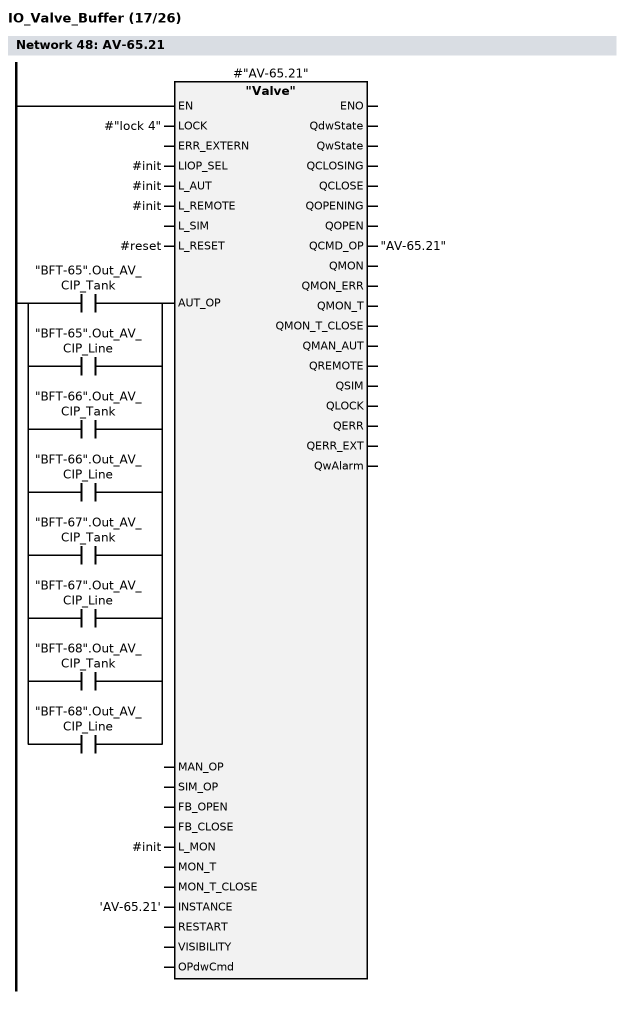
   RUNG wire#powerrail
      #"AV-65.21"(AUT_OP := wire#w1, LOCK := #"lock 4", ERR_EXTERN :=, LIOP_SEL := #init, L_AUT := #init, L_REMOTE := #init, L_SIM :=, L_RESET := #reset, MAN_OP :=, SIM_OP :=, FB_OPEN :=, FB_CLOSE :=, L_MON := #init, MON_T :=, MON_T_CLOSE :=, INSTANCE := 'AV-65.21', RESTART :=, VISIBILITY :=, OPdwCmd :=, QdwState =>, QwState =>, QCLOSING =>, QCLOSE =>, QOPENING =>, QOPEN =>, QCMD_OP => "AV-65.21", QMON =>, QMON_ERR =>, QMON_T =>, QMON_T_CLOSE =>, QMAN_AUT =>, QREMOTE =>, QSIM =>, QLOCK =>, QERR =>, QERR_EXT =>, QwAlarm =>)
   END_RUNG
   RUNG wire#powerrail
      Contact( "BFT-65".Out_AV_CIP_Tank )
   END_RUNG wire#w1
   RUNG wire#powerrail
      Contact( "BFT-65".Out_AV_CIP_Line )
   END_RUNG wire#w1
   RUNG wire#powerrail
      Contact( "BFT-66".Out_AV_CIP_Tank )
   END_RUNG wire#w1
   RUNG wire#powerrail
      Contact( "BFT-66".Out_AV_CIP_Line )
   END_RUNG wire#w1
   RUNG wire#powerrail
      Contact( "BFT-67".Out_AV_CIP_Tank )
   END_RUNG wire#w1
   RUNG wire#powerrail
      Contact( "BFT-67".Out_AV_CIP_Line )
   END_RUNG wire#w1
   RUNG wire#powerrail
      Contact( "BFT-68".Out_AV_CIP_Tank )
   END_RUNG wire#w1
   RUNG wire#powerrail
      Contact( "BFT-68".Out_AV_CIP_Line )
   END_RUNG wire#w1
   // the same network as SCL:
   #"AV-65.21"(LOCK := #"lock 4",   // "Valve"
               LIOP_SEL := #init,
               L_AUT := #init,
               L_REMOTE := #init,
               L_RESET := #reset,
               AUT_OP := "BFT-65".Out_AV_CIP_Tank OR "BFT-65".Out_AV_CIP_Line OR "BFT-66".Out_AV_CIP_Tank OR "BFT-66".Out_AV_CIP_Line OR "BFT-67".Out_AV_CIP_Tank OR "BFT-67".Out_AV_CIP_Line OR "BFT-68".Out_AV_CIP_Tank OR "BFT-68".Out_AV_CIP_Line,
               L_MON := #init,
               INSTANCE := 'AV-65.21',
               QCMD_OP => "AV-65.21");
END_REGION

REGION Network 50 (SCL): FB OPEN AND CLOSE VALVE T-66
   IF #testing THEN
       // Statement section IF
       #"AV-66.01".FB_OPEN := #"AV-66.01".QCMD_OP;
       #"AV-66.01".FB_CLOSE := NOT #"AV-66.01".QCMD_OP;
       #"AV-66.02".FB_OPEN := #"AV-66.02".QCMD_OP;
       #"AV-66.02".FB_CLOSE := NOT #"AV-66.02".QCMD_OP;
       #"AV-66.03".FB_OPEN := #"AV-66.03".QCMD_OP;
       #"AV-66.03".FB_CLOSE := NOT #"AV-66.03".QCMD_OP;
       #"AV-66.04".FB_OPEN := #"AV-66.04".QCMD_OP;
       #"AV-66.04".FB_CLOSE := NOT #"AV-66.04".QCMD_OP;
       #"AV-66.05".FB_OPEN := #"AV-66.05".QCMD_OP;
       #"AV-66.05".FB_CLOSE := NOT #"AV-66.05".QCMD_OP;
       #"AV-66.06".FB_OPEN := #"AV-66.06".QCMD_OP;
       #"AV-66.06".FB_CLOSE := NOT #"AV-66.06".QCMD_OP;
   ELSE
       // Statement section ELSE
       #"AV-66.01".FB_OPEN := NOT "ZSC-66.01";
       #"AV-66.01".FB_CLOSE := "ZSC-66.01";
       #"AV-66.02".FB_OPEN := #"AV-66.02".QCMD_OP;
       #"AV-66.02".FB_CLOSE := NOT #"AV-66.02".QCMD_OP;
       #"AV-66.03".FB_OPEN := NOT "ZSC-66.03";
       #"AV-66.03".FB_CLOSE := "ZSC-66.03";
       #"AV-66.04".FB_OPEN := #"AV-66.04".QCMD_OP;
       #"AV-66.04".FB_CLOSE := NOT #"AV-66.04".QCMD_OP;
       #"AV-66.05".FB_OPEN := #"AV-66.05".QCMD_OP;
       #"AV-66.05".FB_CLOSE := NOT #"AV-66.05".QCMD_OP;
       #"AV-66.06".FB_OPEN := NOT "ZSC-66.06";
       #"AV-66.06".FB_CLOSE := "ZSC-66.06";
   END_IF;
END_REGION

NETWORK
TITLE = FB MONITORING TIME VALVE T-66
// FB OPEN TIME
      L     T#20s;
      T     #"AV-66.01".MON_T;
      T     #"AV-66.02".MON_T;
      T     #"AV-66.03".MON_T;
      T     #"AV-66.04".MON_T;
      T     #"AV-66.05".MON_T;
      T     #"AV-66.06".MON_T;
// FB CLOSE TIME
      L     T#20s;
      T     #"AV-66.01".MON_T_CLOSE;
      T     #"AV-66.02".MON_T_CLOSE;
      T     #"AV-66.03".MON_T_CLOSE;
      T     #"AV-66.04".MON_T_CLOSE;
      T     #"AV-66.05".MON_T_CLOSE;
      T     #"AV-66.06".MON_T_CLOSE;

REGION Network 52: AV-66.01 w ZSC
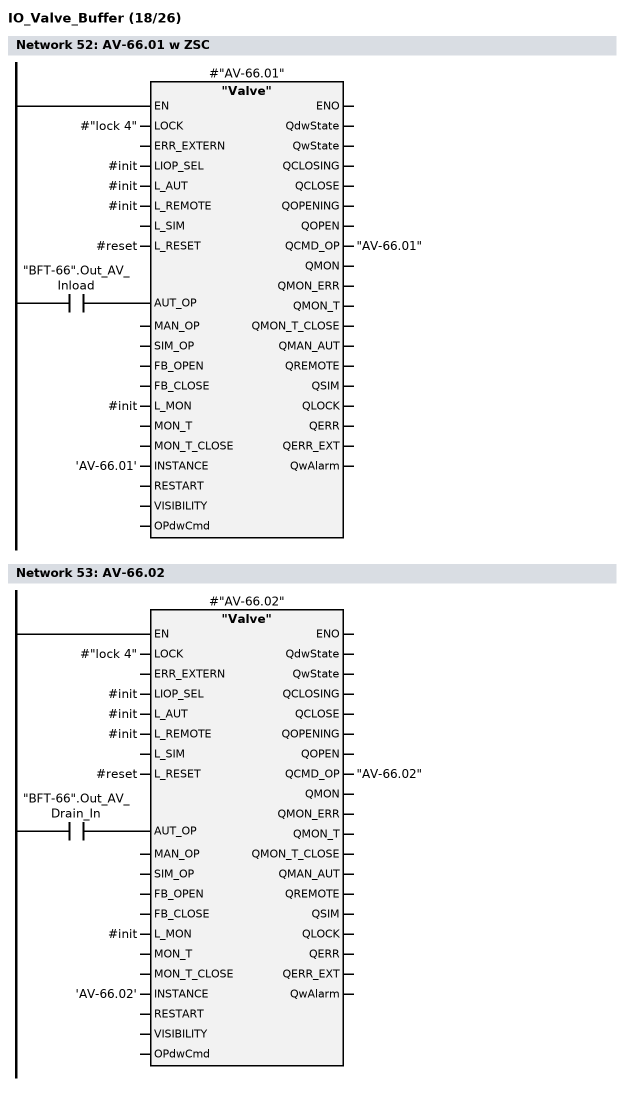
   RUNG wire#powerrail
      #"AV-66.01"(AUT_OP := wire#w1, LOCK := #"lock 4", ERR_EXTERN :=, LIOP_SEL := #init, L_AUT := #init, L_REMOTE := #init, L_SIM :=, L_RESET := #reset, MAN_OP :=, SIM_OP :=, FB_OPEN :=, FB_CLOSE :=, L_MON := #init, MON_T :=, MON_T_CLOSE :=, INSTANCE := 'AV-66.01', RESTART :=, VISIBILITY :=, OPdwCmd :=, QdwState =>, QwState =>, QCLOSING =>, QCLOSE =>, QOPENING =>, QOPEN =>, QCMD_OP => "AV-66.01", QMON =>, QMON_ERR =>, QMON_T =>, QMON_T_CLOSE =>, QMAN_AUT =>, QREMOTE =>, QSIM =>, QLOCK =>, QERR =>, QERR_EXT =>, QwAlarm =>)
   END_RUNG
   RUNG wire#powerrail
      Contact( "BFT-66".Out_AV_Inload )
   END_RUNG wire#w1
   // the same network as SCL:
   #"AV-66.01"(LOCK := #"lock 4",   // "Valve"
               LIOP_SEL := #init,
               L_AUT := #init,
               L_REMOTE := #init,
               L_RESET := #reset,
               AUT_OP := "BFT-66".Out_AV_Inload,
               L_MON := #init,
               INSTANCE := 'AV-66.01',
               QCMD_OP => "AV-66.01");
END_REGION

REGION Network 53: AV-66.02
   RUNG wire#powerrail
      #"AV-66.02"(AUT_OP := wire#w1, LOCK := #"lock 4", ERR_EXTERN :=, LIOP_SEL := #init, L_AUT := #init, L_REMOTE := #init, L_SIM :=, L_RESET := #reset, MAN_OP :=, SIM_OP :=, FB_OPEN :=, FB_CLOSE :=, L_MON := #init, MON_T :=, MON_T_CLOSE :=, INSTANCE := 'AV-66.02', RESTART :=, VISIBILITY :=, OPdwCmd :=, QdwState =>, QwState =>, QCLOSING =>, QCLOSE =>, QOPENING =>, QOPEN =>, QCMD_OP => "AV-66.02", QMON =>, QMON_ERR =>, QMON_T =>, QMON_T_CLOSE =>, QMAN_AUT =>, QREMOTE =>, QSIM =>, QLOCK =>, QERR =>, QERR_EXT =>, QwAlarm =>)
   END_RUNG
   RUNG wire#powerrail
      Contact( "BFT-66".Out_AV_Drain_In )
   END_RUNG wire#w1
   // the same network as SCL:
   #"AV-66.02"(LOCK := #"lock 4",   // "Valve"
               LIOP_SEL := #init,
               L_AUT := #init,
               L_REMOTE := #init,
               L_RESET := #reset,
               AUT_OP := "BFT-66".Out_AV_Drain_In,
               L_MON := #init,
               INSTANCE := 'AV-66.02',
               QCMD_OP => "AV-66.02");
END_REGION

REGION Network 54: AV-66.03 w ZSC
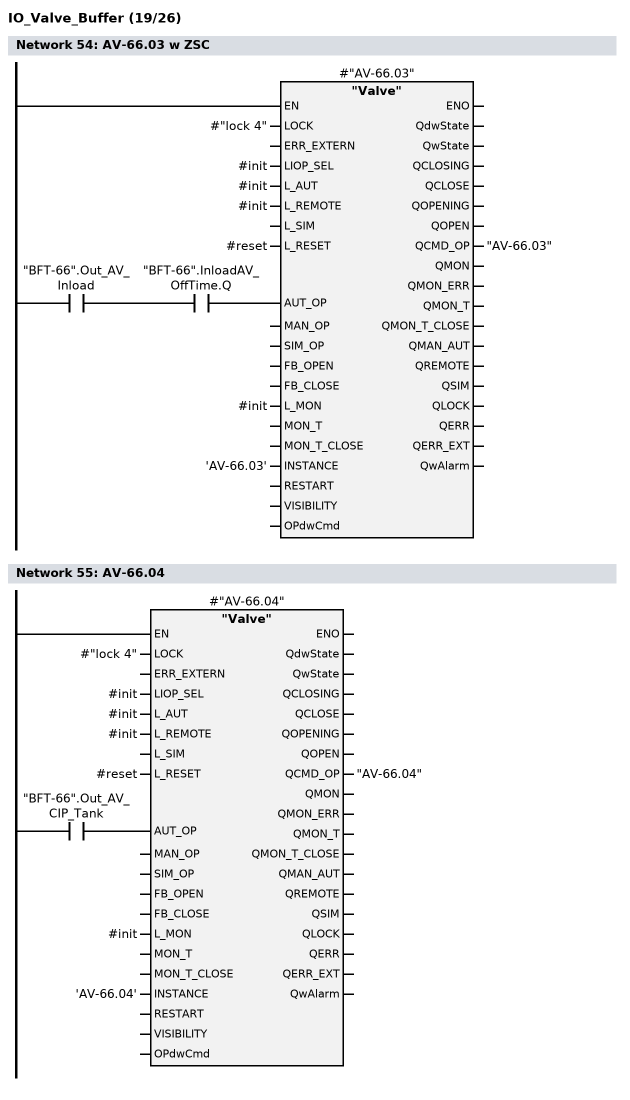
   RUNG wire#powerrail
      #"AV-66.03"(AUT_OP := wire#w1, LOCK := #"lock 4", ERR_EXTERN :=, LIOP_SEL := #init, L_AUT := #init, L_REMOTE := #init, L_SIM :=, L_RESET := #reset, MAN_OP :=, SIM_OP :=, FB_OPEN :=, FB_CLOSE :=, L_MON := #init, MON_T :=, MON_T_CLOSE :=, INSTANCE := 'AV-66.03', RESTART :=, VISIBILITY :=, OPdwCmd :=, QdwState =>, QwState =>, QCLOSING =>, QCLOSE =>, QOPENING =>, QOPEN =>, QCMD_OP => "AV-66.03", QMON =>, QMON_ERR =>, QMON_T =>, QMON_T_CLOSE =>, QMAN_AUT =>, QREMOTE =>, QSIM =>, QLOCK =>, QERR =>, QERR_EXT =>, QwAlarm =>)
   END_RUNG
   RUNG wire#powerrail
      Contact( "BFT-66".Out_AV_Inload )
      Contact( "BFT-66".InloadAV_OffTime.Q )
   END_RUNG wire#w1
   // the same network as SCL:
   #"AV-66.03"(LOCK := #"lock 4",   // "Valve"
               LIOP_SEL := #init,
               L_AUT := #init,
               L_REMOTE := #init,
               L_RESET := #reset,
               AUT_OP := "BFT-66".Out_AV_Inload AND "BFT-66".InloadAV_OffTime.Q,
               L_MON := #init,
               INSTANCE := 'AV-66.03',
               QCMD_OP => "AV-66.03");
END_REGION

REGION Network 55: AV-66.04
   RUNG wire#powerrail
      #"AV-66.04"(AUT_OP := wire#w1, LOCK := #"lock 4", ERR_EXTERN :=, LIOP_SEL := #init, L_AUT := #init, L_REMOTE := #init, L_SIM :=, L_RESET := #reset, MAN_OP :=, SIM_OP :=, FB_OPEN :=, FB_CLOSE :=, L_MON := #init, MON_T :=, MON_T_CLOSE :=, INSTANCE := 'AV-66.04', RESTART :=, VISIBILITY :=, OPdwCmd :=, QdwState =>, QwState =>, QCLOSING =>, QCLOSE =>, QOPENING =>, QOPEN =>, QCMD_OP => "AV-66.04", QMON =>, QMON_ERR =>, QMON_T =>, QMON_T_CLOSE =>, QMAN_AUT =>, QREMOTE =>, QSIM =>, QLOCK =>, QERR =>, QERR_EXT =>, QwAlarm =>)
   END_RUNG
   RUNG wire#powerrail
      Contact( "BFT-66".Out_AV_CIP_Tank )
   END_RUNG wire#w1
   // the same network as SCL:
   #"AV-66.04"(LOCK := #"lock 4",   // "Valve"
               LIOP_SEL := #init,
               L_AUT := #init,
               L_REMOTE := #init,
               L_RESET := #reset,
               AUT_OP := "BFT-66".Out_AV_CIP_Tank,
               L_MON := #init,
               INSTANCE := 'AV-66.04',
               QCMD_OP => "AV-66.04");
END_REGION

REGION Network 56: AV-66.05
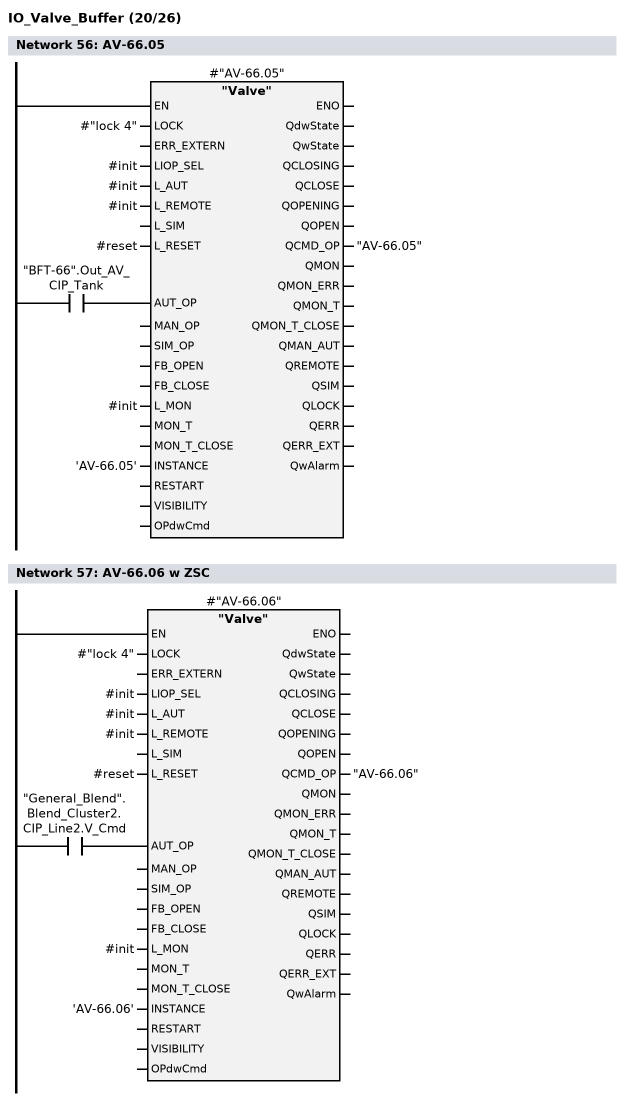
   RUNG wire#powerrail
      #"AV-66.05"(AUT_OP := wire#w1, LOCK := #"lock 4", ERR_EXTERN :=, LIOP_SEL := #init, L_AUT := #init, L_REMOTE := #init, L_SIM :=, L_RESET := #reset, MAN_OP :=, SIM_OP :=, FB_OPEN :=, FB_CLOSE :=, L_MON := #init, MON_T :=, MON_T_CLOSE :=, INSTANCE := 'AV-66.05', RESTART :=, VISIBILITY :=, OPdwCmd :=, QdwState =>, QwState =>, QCLOSING =>, QCLOSE =>, QOPENING =>, QOPEN =>, QCMD_OP => "AV-66.05", QMON =>, QMON_ERR =>, QMON_T =>, QMON_T_CLOSE =>, QMAN_AUT =>, QREMOTE =>, QSIM =>, QLOCK =>, QERR =>, QERR_EXT =>, QwAlarm =>)
   END_RUNG
   RUNG wire#powerrail
      Contact( "BFT-66".Out_AV_CIP_Tank )
   END_RUNG wire#w1
   // the same network as SCL:
   #"AV-66.05"(LOCK := #"lock 4",   // "Valve"
               LIOP_SEL := #init,
               L_AUT := #init,
               L_REMOTE := #init,
               L_RESET := #reset,
               AUT_OP := "BFT-66".Out_AV_CIP_Tank,
               L_MON := #init,
               INSTANCE := 'AV-66.05',
               QCMD_OP => "AV-66.05");
END_REGION

REGION Network 57: AV-66.06 w ZSC
   RUNG wire#powerrail
      #"AV-66.06"(AUT_OP := wire#w1, LOCK := #"lock 4", ERR_EXTERN :=, LIOP_SEL := #init, L_AUT := #init, L_REMOTE := #init, L_SIM :=, L_RESET := #reset, MAN_OP :=, SIM_OP :=, FB_OPEN :=, FB_CLOSE :=, L_MON := #init, MON_T :=, MON_T_CLOSE :=, INSTANCE := 'AV-66.06', RESTART :=, VISIBILITY :=, OPdwCmd :=, QdwState =>, QwState =>, QCLOSING =>, QCLOSE =>, QOPENING =>, QOPEN =>, QCMD_OP => "AV-66.06", QMON =>, QMON_ERR =>, QMON_T =>, QMON_T_CLOSE =>, QMAN_AUT =>, QREMOTE =>, QSIM =>, QLOCK =>, QERR =>, QERR_EXT =>, QwAlarm =>)
   END_RUNG
   RUNG wire#powerrail
      Contact( "General_Blend".Blend_Cluster2.CIP_Line2.V_Cmd )
   END_RUNG wire#w1
   // the same network as SCL:
   #"AV-66.06"(LOCK := #"lock 4",   // "Valve"
               LIOP_SEL := #init,
               L_AUT := #init,
               L_REMOTE := #init,
               L_RESET := #reset,
               AUT_OP := "General_Blend".Blend_Cluster2.CIP_Line2.V_Cmd,
               L_MON := #init,
               INSTANCE := 'AV-66.06',
               QCMD_OP => "AV-66.06");
END_REGION

REGION Network 59 (SCL): FB OPEN AND CLOSE VALVE T-67
   IF #testing THEN
       // Statement section IF
       #"AV-67.01".FB_OPEN := #"AV-67.01".QCMD_OP;
       #"AV-67.01".FB_CLOSE := NOT #"AV-67.01".QCMD_OP;
       #"AV-67.02".FB_OPEN := #"AV-67.02".QCMD_OP;
       #"AV-67.02".FB_CLOSE := NOT #"AV-67.02".QCMD_OP;
       #"AV-67.03".FB_OPEN := #"AV-67.03".QCMD_OP;
       #"AV-67.03".FB_CLOSE := NOT #"AV-67.03".QCMD_OP;
       #"AV-67.04".FB_OPEN := #"AV-67.04".QCMD_OP;
       #"AV-67.04".FB_CLOSE := NOT #"AV-67.04".QCMD_OP;
       #"AV-67.05".FB_OPEN := #"AV-67.05".QCMD_OP;
       #"AV-67.05".FB_CLOSE := NOT #"AV-67.05".QCMD_OP;
   ELSE
       // Statement section ELSE
       #"AV-67.01".FB_OPEN := NOT "ZSC-67.01";
       #"AV-67.01".FB_CLOSE := "ZSC-67.01";
       #"AV-67.02".FB_OPEN := #"AV-67.02".QCMD_OP;
       #"AV-67.02".FB_CLOSE := NOT #"AV-67.02".QCMD_OP;
       #"AV-67.03".FB_OPEN := NOT "ZSC-67.03";
       #"AV-67.03".FB_CLOSE := "ZSC-67.03";
       #"AV-67.04".FB_OPEN := #"AV-67.04".QCMD_OP;
       #"AV-67.04".FB_CLOSE := NOT #"AV-67.04".QCMD_OP;
       #"AV-67.05".FB_OPEN := #"AV-67.05".QCMD_OP;
       #"AV-67.05".FB_CLOSE := NOT #"AV-67.05".QCMD_OP;
   END_IF;
END_REGION

NETWORK
TITLE = FB MONITORING TIME VALVE T-67
// FB OPEN TIME
      L     T#20s;
      T     #"AV-67.01".MON_T;
      T     #"AV-67.02".MON_T;
      T     #"AV-67.03".MON_T;
      T     #"AV-67.04".MON_T;
      T     #"AV-67.05".MON_T;
// FB CLOSE TIME
      L     T#20s;
      T     #"AV-67.01".MON_T_CLOSE;
      T     #"AV-67.02".MON_T_CLOSE;
      T     #"AV-67.03".MON_T_CLOSE;
      T     #"AV-67.04".MON_T_CLOSE;
      T     #"AV-67.05".MON_T_CLOSE;


REGION Network 61: AV-67.01 w ZSC
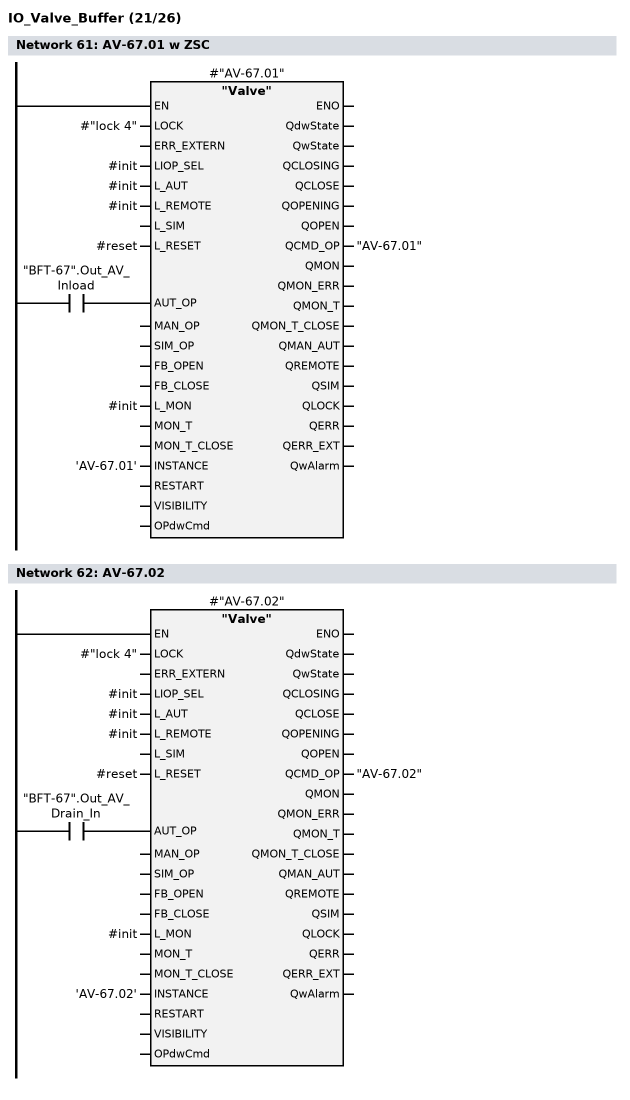
   RUNG wire#powerrail
      #"AV-67.01"(AUT_OP := wire#w1, LOCK := #"lock 4", ERR_EXTERN :=, LIOP_SEL := #init, L_AUT := #init, L_REMOTE := #init, L_SIM :=, L_RESET := #reset, MAN_OP :=, SIM_OP :=, FB_OPEN :=, FB_CLOSE :=, L_MON := #init, MON_T :=, MON_T_CLOSE :=, INSTANCE := 'AV-67.01', RESTART :=, VISIBILITY :=, OPdwCmd :=, QdwState =>, QwState =>, QCLOSING =>, QCLOSE =>, QOPENING =>, QOPEN =>, QCMD_OP => "AV-67.01", QMON =>, QMON_ERR =>, QMON_T =>, QMON_T_CLOSE =>, QMAN_AUT =>, QREMOTE =>, QSIM =>, QLOCK =>, QERR =>, QERR_EXT =>, QwAlarm =>)
   END_RUNG
   RUNG wire#powerrail
      Contact( "BFT-67".Out_AV_Inload )
   END_RUNG wire#w1
   // the same network as SCL:
   #"AV-67.01"(LOCK := #"lock 4",   // "Valve"
               LIOP_SEL := #init,
               L_AUT := #init,
               L_REMOTE := #init,
               L_RESET := #reset,
               AUT_OP := "BFT-67".Out_AV_Inload,
               L_MON := #init,
               INSTANCE := 'AV-67.01',
               QCMD_OP => "AV-67.01");
END_REGION

REGION Network 62: AV-67.02
   RUNG wire#powerrail
      #"AV-67.02"(AUT_OP := wire#w1, LOCK := #"lock 4", ERR_EXTERN :=, LIOP_SEL := #init, L_AUT := #init, L_REMOTE := #init, L_SIM :=, L_RESET := #reset, MAN_OP :=, SIM_OP :=, FB_OPEN :=, FB_CLOSE :=, L_MON := #init, MON_T :=, MON_T_CLOSE :=, INSTANCE := 'AV-67.02', RESTART :=, VISIBILITY :=, OPdwCmd :=, QdwState =>, QwState =>, QCLOSING =>, QCLOSE =>, QOPENING =>, QOPEN =>, QCMD_OP => "AV-67.02", QMON =>, QMON_ERR =>, QMON_T =>, QMON_T_CLOSE =>, QMAN_AUT =>, QREMOTE =>, QSIM =>, QLOCK =>, QERR =>, QERR_EXT =>, QwAlarm =>)
   END_RUNG
   RUNG wire#powerrail
      Contact( "BFT-67".Out_AV_Drain_In )
   END_RUNG wire#w1
   // the same network as SCL:
   #"AV-67.02"(LOCK := #"lock 4",   // "Valve"
               LIOP_SEL := #init,
               L_AUT := #init,
               L_REMOTE := #init,
               L_RESET := #reset,
               AUT_OP := "BFT-67".Out_AV_Drain_In,
               L_MON := #init,
               INSTANCE := 'AV-67.02',
               QCMD_OP => "AV-67.02");
END_REGION

REGION Network 63: AV-67.03 w ZSC
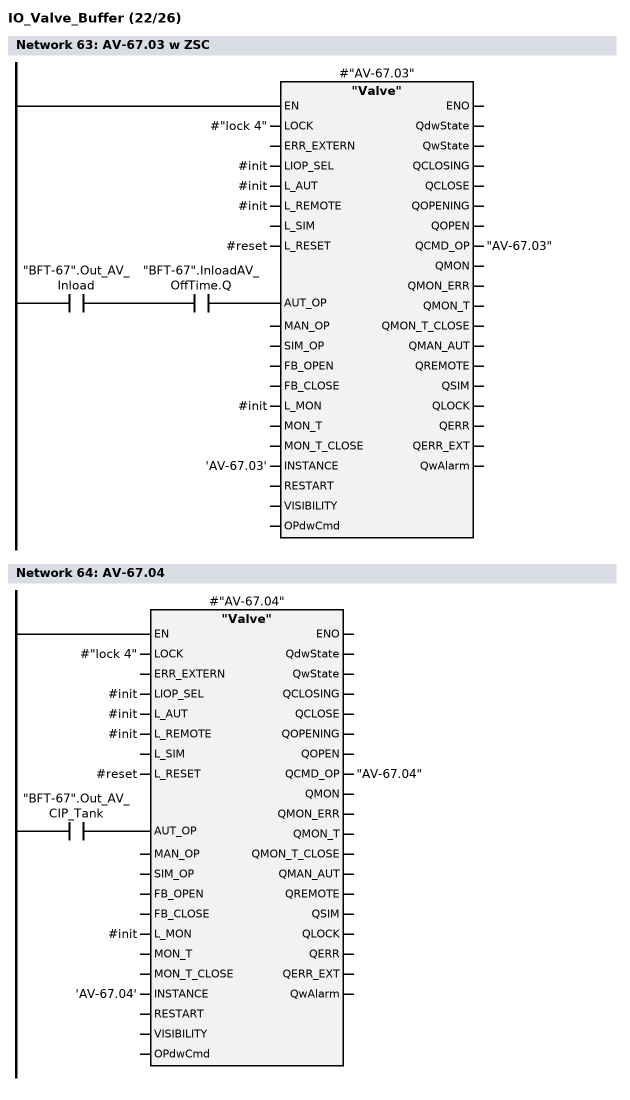
   RUNG wire#powerrail
      #"AV-67.03"(AUT_OP := wire#w1, LOCK := #"lock 4", ERR_EXTERN :=, LIOP_SEL := #init, L_AUT := #init, L_REMOTE := #init, L_SIM :=, L_RESET := #reset, MAN_OP :=, SIM_OP :=, FB_OPEN :=, FB_CLOSE :=, L_MON := #init, MON_T :=, MON_T_CLOSE :=, INSTANCE := 'AV-67.03', RESTART :=, VISIBILITY :=, OPdwCmd :=, QdwState =>, QwState =>, QCLOSING =>, QCLOSE =>, QOPENING =>, QOPEN =>, QCMD_OP => "AV-67.03", QMON =>, QMON_ERR =>, QMON_T =>, QMON_T_CLOSE =>, QMAN_AUT =>, QREMOTE =>, QSIM =>, QLOCK =>, QERR =>, QERR_EXT =>, QwAlarm =>)
   END_RUNG
   RUNG wire#powerrail
      Contact( "BFT-67".Out_AV_Inload )
      Contact( "BFT-67".InloadAV_OffTime.Q )
   END_RUNG wire#w1
   // the same network as SCL:
   #"AV-67.03"(LOCK := #"lock 4",   // "Valve"
               LIOP_SEL := #init,
               L_AUT := #init,
               L_REMOTE := #init,
               L_RESET := #reset,
               AUT_OP := "BFT-67".Out_AV_Inload AND "BFT-67".InloadAV_OffTime.Q,
               L_MON := #init,
               INSTANCE := 'AV-67.03',
               QCMD_OP => "AV-67.03");
END_REGION

REGION Network 64: AV-67.04
   RUNG wire#powerrail
      #"AV-67.04"(AUT_OP := wire#w1, LOCK := #"lock 4", ERR_EXTERN :=, LIOP_SEL := #init, L_AUT := #init, L_REMOTE := #init, L_SIM :=, L_RESET := #reset, MAN_OP :=, SIM_OP :=, FB_OPEN :=, FB_CLOSE :=, L_MON := #init, MON_T :=, MON_T_CLOSE :=, INSTANCE := 'AV-67.04', RESTART :=, VISIBILITY :=, OPdwCmd :=, QdwState =>, QwState =>, QCLOSING =>, QCLOSE =>, QOPENING =>, QOPEN =>, QCMD_OP => "AV-67.04", QMON =>, QMON_ERR =>, QMON_T =>, QMON_T_CLOSE =>, QMAN_AUT =>, QREMOTE =>, QSIM =>, QLOCK =>, QERR =>, QERR_EXT =>, QwAlarm =>)
   END_RUNG
   RUNG wire#powerrail
      Contact( "BFT-67".Out_AV_CIP_Tank )
   END_RUNG wire#w1
   // the same network as SCL:
   #"AV-67.04"(LOCK := #"lock 4",   // "Valve"
               LIOP_SEL := #init,
               L_AUT := #init,
               L_REMOTE := #init,
               L_RESET := #reset,
               AUT_OP := "BFT-67".Out_AV_CIP_Tank,
               L_MON := #init,
               INSTANCE := 'AV-67.04',
               QCMD_OP => "AV-67.04");
END_REGION

REGION Network 65: AV-67.05
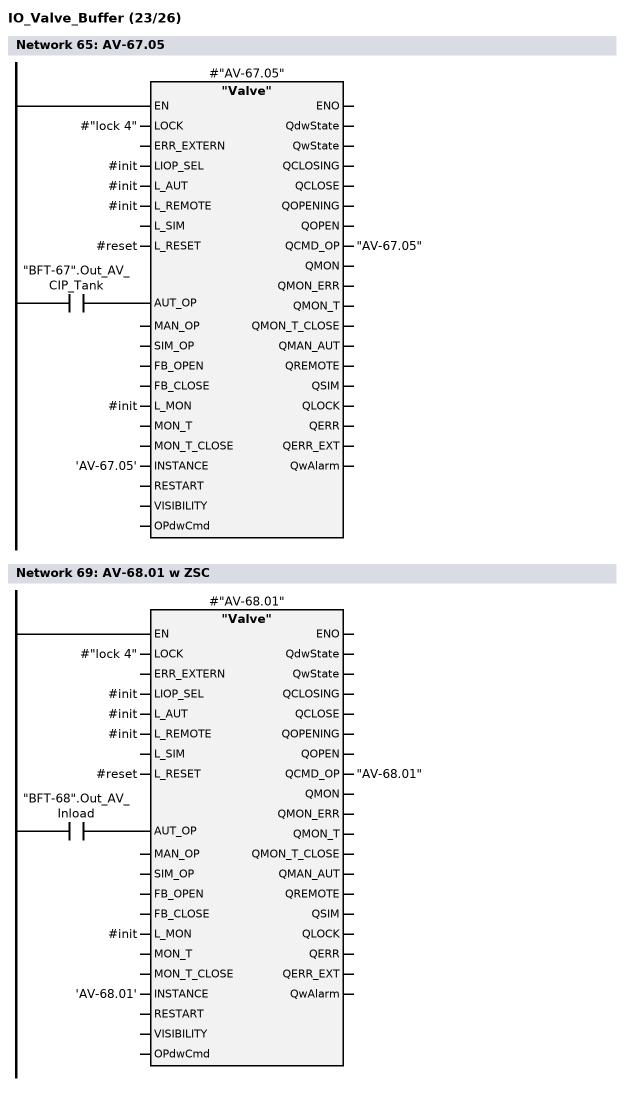
   RUNG wire#powerrail
      #"AV-67.05"(AUT_OP := wire#w1, LOCK := #"lock 4", ERR_EXTERN :=, LIOP_SEL := #init, L_AUT := #init, L_REMOTE := #init, L_SIM :=, L_RESET := #reset, MAN_OP :=, SIM_OP :=, FB_OPEN :=, FB_CLOSE :=, L_MON := #init, MON_T :=, MON_T_CLOSE :=, INSTANCE := 'AV-67.05', RESTART :=, VISIBILITY :=, OPdwCmd :=, QdwState =>, QwState =>, QCLOSING =>, QCLOSE =>, QOPENING =>, QOPEN =>, QCMD_OP => "AV-67.05", QMON =>, QMON_ERR =>, QMON_T =>, QMON_T_CLOSE =>, QMAN_AUT =>, QREMOTE =>, QSIM =>, QLOCK =>, QERR =>, QERR_EXT =>, QwAlarm =>)
   END_RUNG
   RUNG wire#powerrail
      Contact( "BFT-67".Out_AV_CIP_Tank )
   END_RUNG wire#w1
   // the same network as SCL:
   #"AV-67.05"(LOCK := #"lock 4",   // "Valve"
               LIOP_SEL := #init,
               L_AUT := #init,
               L_REMOTE := #init,
               L_RESET := #reset,
               AUT_OP := "BFT-67".Out_AV_CIP_Tank,
               L_MON := #init,
               INSTANCE := 'AV-67.05',
               QCMD_OP => "AV-67.05");
END_REGION

REGION Network 67 (SCL): FB OPEN AND CLOSE VALVE T-68
   IF #testing THEN
       // Statement section IF
       #"AV-68.01".FB_OPEN := #"AV-68.01".QCMD_OP;
       #"AV-68.01".FB_CLOSE := NOT #"AV-68.01".QCMD_OP;
       #"AV-68.02".FB_OPEN := #"AV-68.02".QCMD_OP;
       #"AV-68.02".FB_CLOSE := NOT #"AV-68.02".QCMD_OP;
       #"AV-68.03".FB_OPEN := #"AV-68.03".QCMD_OP;
       #"AV-68.03".FB_CLOSE := NOT #"AV-68.03".QCMD_OP;
       #"AV-68.04".FB_OPEN := #"AV-68.04".QCMD_OP;
       #"AV-68.04".FB_CLOSE := NOT #"AV-68.04".QCMD_OP;
       #"AV-68.05".FB_OPEN := #"AV-68.05".QCMD_OP;
       #"AV-68.05".FB_CLOSE := NOT #"AV-68.05".QCMD_OP;
       #"AV-68.06".FB_OPEN := #"AV-68.06".QCMD_OP;
       #"AV-68.06".FB_CLOSE := NOT #"AV-68.06".QCMD_OP;
   ELSE
       // Statement section ELSE
       #"AV-68.01".FB_OPEN := NOT "ZSC-68.01";
       #"AV-68.01".FB_CLOSE := "ZSC-68.01";
       #"AV-68.02".FB_OPEN := #"AV-68.02".QCMD_OP;
       #"AV-68.02".FB_CLOSE := NOT #"AV-68.02".QCMD_OP;
       #"AV-68.03".FB_OPEN := NOT "ZSC-68.03";
       #"AV-68.03".FB_CLOSE := "ZSC-68.03";
       #"AV-68.04".FB_OPEN := #"AV-68.04".QCMD_OP;
       #"AV-68.04".FB_CLOSE := NOT #"AV-68.04".QCMD_OP;
       #"AV-68.05".FB_OPEN := #"AV-68.05".QCMD_OP;
       #"AV-68.05".FB_CLOSE := NOT #"AV-68.05".QCMD_OP;
       #"AV-68.06".FB_OPEN := NOT "ZSC-68.06";
       #"AV-68.06".FB_CLOSE := "ZSC-68.06";
   END_IF;
END_REGION

NETWORK
TITLE = FB MONITORING TIME VALVE T-68
// FB OPEN TIME
      L     T#20s;
      T     #"AV-68.01".MON_T;
      T     #"AV-68.02".MON_T;
      T     #"AV-68.03".MON_T;
      T     #"AV-68.04".MON_T;
      T     #"AV-68.05".MON_T;
      T     #"AV-68.06".MON_T;
// FB CLOSE TIME
      L     T#20s;
      T     #"AV-68.01".MON_T_CLOSE;
      T     #"AV-68.02".MON_T_CLOSE;
      T     #"AV-68.03".MON_T_CLOSE;
      T     #"AV-68.04".MON_T_CLOSE;
      T     #"AV-68.05".MON_T_CLOSE;
      T     #"AV-68.06".MON_T_CLOSE;

REGION Network 69: AV-68.01 w ZSC
   RUNG wire#powerrail
      #"AV-68.01"(AUT_OP := wire#w1, LOCK := #"lock 4", ERR_EXTERN :=, LIOP_SEL := #init, L_AUT := #init, L_REMOTE := #init, L_SIM :=, L_RESET := #reset, MAN_OP :=, SIM_OP :=, FB_OPEN :=, FB_CLOSE :=, L_MON := #init, MON_T :=, MON_T_CLOSE :=, INSTANCE := 'AV-68.01', RESTART :=, VISIBILITY :=, OPdwCmd :=, QdwState =>, QwState =>, QCLOSING =>, QCLOSE =>, QOPENING =>, QOPEN =>, QCMD_OP => "AV-68.01", QMON =>, QMON_ERR =>, QMON_T =>, QMON_T_CLOSE =>, QMAN_AUT =>, QREMOTE =>, QSIM =>, QLOCK =>, QERR =>, QERR_EXT =>, QwAlarm =>)
   END_RUNG
   RUNG wire#powerrail
      Contact( "BFT-68".Out_AV_Inload )
   END_RUNG wire#w1
   // the same network as SCL:
   #"AV-68.01"(LOCK := #"lock 4",   // "Valve"
               LIOP_SEL := #init,
               L_AUT := #init,
               L_REMOTE := #init,
               L_RESET := #reset,
               AUT_OP := "BFT-68".Out_AV_Inload,
               L_MON := #init,
               INSTANCE := 'AV-68.01',
               QCMD_OP => "AV-68.01");
END_REGION

REGION Network 70: AV-68.02
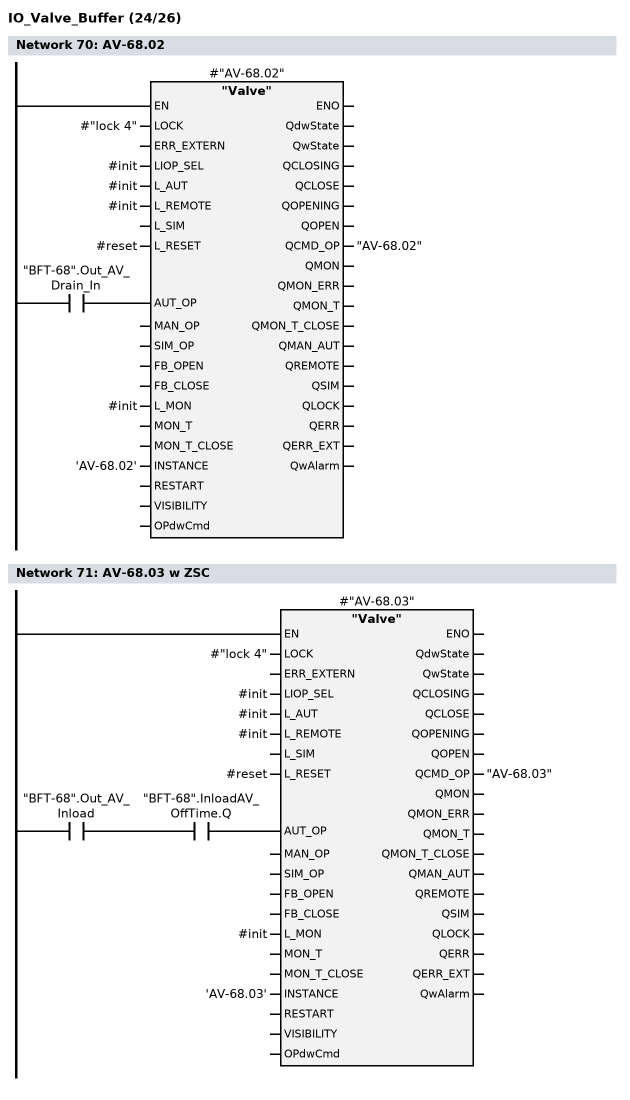
   RUNG wire#powerrail
      #"AV-68.02"(AUT_OP := wire#w1, LOCK := #"lock 4", ERR_EXTERN :=, LIOP_SEL := #init, L_AUT := #init, L_REMOTE := #init, L_SIM :=, L_RESET := #reset, MAN_OP :=, SIM_OP :=, FB_OPEN :=, FB_CLOSE :=, L_MON := #init, MON_T :=, MON_T_CLOSE :=, INSTANCE := 'AV-68.02', RESTART :=, VISIBILITY :=, OPdwCmd :=, QdwState =>, QwState =>, QCLOSING =>, QCLOSE =>, QOPENING =>, QOPEN =>, QCMD_OP => "AV-68.02", QMON =>, QMON_ERR =>, QMON_T =>, QMON_T_CLOSE =>, QMAN_AUT =>, QREMOTE =>, QSIM =>, QLOCK =>, QERR =>, QERR_EXT =>, QwAlarm =>)
   END_RUNG
   RUNG wire#powerrail
      Contact( "BFT-68".Out_AV_Drain_In )
   END_RUNG wire#w1
   // the same network as SCL:
   #"AV-68.02"(LOCK := #"lock 4",   // "Valve"
               LIOP_SEL := #init,
               L_AUT := #init,
               L_REMOTE := #init,
               L_RESET := #reset,
               AUT_OP := "BFT-68".Out_AV_Drain_In,
               L_MON := #init,
               INSTANCE := 'AV-68.02',
               QCMD_OP => "AV-68.02");
END_REGION

REGION Network 71: AV-68.03 w ZSC
   RUNG wire#powerrail
      #"AV-68.03"(AUT_OP := wire#w1, LOCK := #"lock 4", ERR_EXTERN :=, LIOP_SEL := #init, L_AUT := #init, L_REMOTE := #init, L_SIM :=, L_RESET := #reset, MAN_OP :=, SIM_OP :=, FB_OPEN :=, FB_CLOSE :=, L_MON := #init, MON_T :=, MON_T_CLOSE :=, INSTANCE := 'AV-68.03', RESTART :=, VISIBILITY :=, OPdwCmd :=, QdwState =>, QwState =>, QCLOSING =>, QCLOSE =>, QOPENING =>, QOPEN =>, QCMD_OP => "AV-68.03", QMON =>, QMON_ERR =>, QMON_T =>, QMON_T_CLOSE =>, QMAN_AUT =>, QREMOTE =>, QSIM =>, QLOCK =>, QERR =>, QERR_EXT =>, QwAlarm =>)
   END_RUNG
   RUNG wire#powerrail
      Contact( "BFT-68".Out_AV_Inload )
      Contact( "BFT-68".InloadAV_OffTime.Q )
   END_RUNG wire#w1
   // the same network as SCL:
   #"AV-68.03"(LOCK := #"lock 4",   // "Valve"
               LIOP_SEL := #init,
               L_AUT := #init,
               L_REMOTE := #init,
               L_RESET := #reset,
               AUT_OP := "BFT-68".Out_AV_Inload AND "BFT-68".InloadAV_OffTime.Q,
               L_MON := #init,
               INSTANCE := 'AV-68.03',
               QCMD_OP => "AV-68.03");
END_REGION

REGION Network 72: AV-68.04
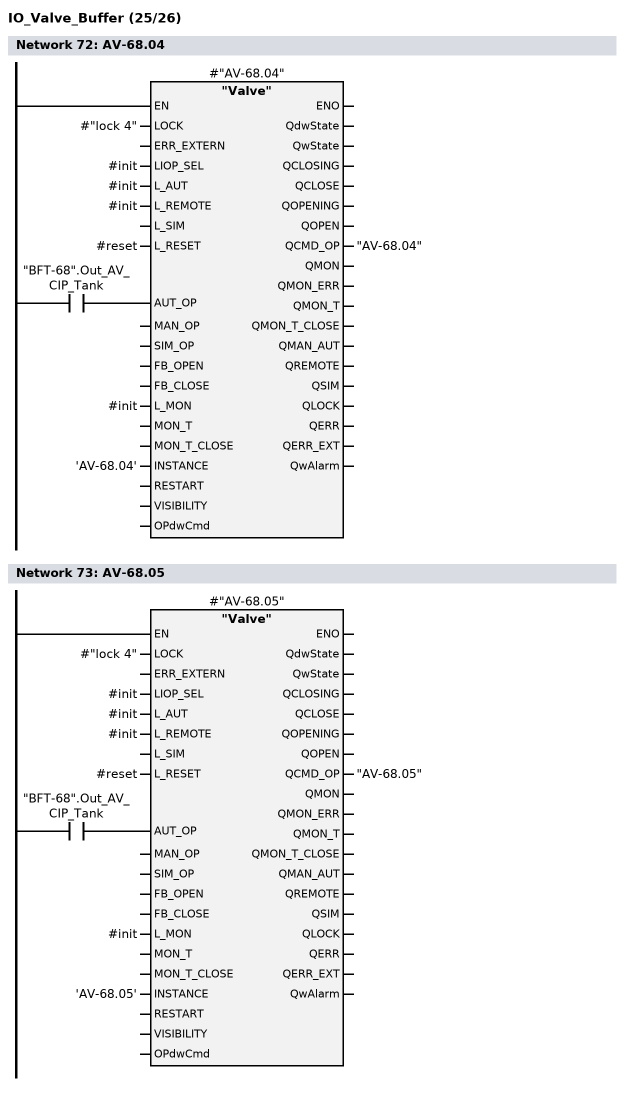
   RUNG wire#powerrail
      #"AV-68.04"(AUT_OP := wire#w1, LOCK := #"lock 4", ERR_EXTERN :=, LIOP_SEL := #init, L_AUT := #init, L_REMOTE := #init, L_SIM :=, L_RESET := #reset, MAN_OP :=, SIM_OP :=, FB_OPEN :=, FB_CLOSE :=, L_MON := #init, MON_T :=, MON_T_CLOSE :=, INSTANCE := 'AV-68.04', RESTART :=, VISIBILITY :=, OPdwCmd :=, QdwState =>, QwState =>, QCLOSING =>, QCLOSE =>, QOPENING =>, QOPEN =>, QCMD_OP => "AV-68.04", QMON =>, QMON_ERR =>, QMON_T =>, QMON_T_CLOSE =>, QMAN_AUT =>, QREMOTE =>, QSIM =>, QLOCK =>, QERR =>, QERR_EXT =>, QwAlarm =>)
   END_RUNG
   RUNG wire#powerrail
      Contact( "BFT-68".Out_AV_CIP_Tank )
   END_RUNG wire#w1
   // the same network as SCL:
   #"AV-68.04"(LOCK := #"lock 4",   // "Valve"
               LIOP_SEL := #init,
               L_AUT := #init,
               L_REMOTE := #init,
               L_RESET := #reset,
               AUT_OP := "BFT-68".Out_AV_CIP_Tank,
               L_MON := #init,
               INSTANCE := 'AV-68.04',
               QCMD_OP => "AV-68.04");
END_REGION

REGION Network 73: AV-68.05
   RUNG wire#powerrail
      #"AV-68.05"(AUT_OP := wire#w1, LOCK := #"lock 4", ERR_EXTERN :=, LIOP_SEL := #init, L_AUT := #init, L_REMOTE := #init, L_SIM :=, L_RESET := #reset, MAN_OP :=, SIM_OP :=, FB_OPEN :=, FB_CLOSE :=, L_MON := #init, MON_T :=, MON_T_CLOSE :=, INSTANCE := 'AV-68.05', RESTART :=, VISIBILITY :=, OPdwCmd :=, QdwState =>, QwState =>, QCLOSING =>, QCLOSE =>, QOPENING =>, QOPEN =>, QCMD_OP => "AV-68.05", QMON =>, QMON_ERR =>, QMON_T =>, QMON_T_CLOSE =>, QMAN_AUT =>, QREMOTE =>, QSIM =>, QLOCK =>, QERR =>, QERR_EXT =>, QwAlarm =>)
   END_RUNG
   RUNG wire#powerrail
      Contact( "BFT-68".Out_AV_CIP_Tank )
   END_RUNG wire#w1
   // the same network as SCL:
   #"AV-68.05"(LOCK := #"lock 4",   // "Valve"
               LIOP_SEL := #init,
               L_AUT := #init,
               L_REMOTE := #init,
               L_RESET := #reset,
               AUT_OP := "BFT-68".Out_AV_CIP_Tank,
               L_MON := #init,
               INSTANCE := 'AV-68.05',
               QCMD_OP => "AV-68.05");
END_REGION

REGION Network 74: AV-68.06 w ZSC
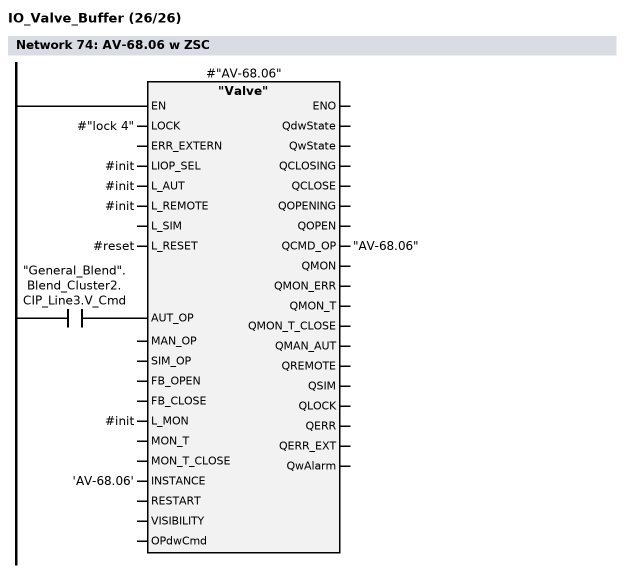
   RUNG wire#powerrail
      #"AV-68.06"(AUT_OP := wire#w1, LOCK := #"lock 4", ERR_EXTERN :=, LIOP_SEL := #init, L_AUT := #init, L_REMOTE := #init, L_SIM :=, L_RESET := #reset, MAN_OP :=, SIM_OP :=, FB_OPEN :=, FB_CLOSE :=, L_MON := #init, MON_T :=, MON_T_CLOSE :=, INSTANCE := 'AV-68.06', RESTART :=, VISIBILITY :=, OPdwCmd :=, QdwState =>, QwState =>, QCLOSING =>, QCLOSE =>, QOPENING =>, QOPEN =>, QCMD_OP => "AV-68.06", QMON =>, QMON_ERR =>, QMON_T =>, QMON_T_CLOSE =>, QMAN_AUT =>, QREMOTE =>, QSIM =>, QLOCK =>, QERR =>, QERR_EXT =>, QwAlarm =>)
   END_RUNG
   RUNG wire#powerrail
      Contact( "General_Blend".Blend_Cluster2.CIP_Line3.V_Cmd )
   END_RUNG wire#w1
   // the same network as SCL:
   #"AV-68.06"(LOCK := #"lock 4",   // "Valve"
               LIOP_SEL := #init,
               L_AUT := #init,
               L_REMOTE := #init,
               L_RESET := #reset,
               AUT_OP := "General_Blend".Blend_Cluster2.CIP_Line3.V_Cmd,
               L_MON := #init,
               INSTANCE := 'AV-68.06',
               QCMD_OP => "AV-68.06");
END_REGION
END_FUNCTION_BLOCK

FUNCTION_BLOCK "Alarm_Collector_Gen"   // FB33, LAD
{ S7_Optimized_Access := 'TRUE' }
VERSION : 0.1
// stored: AutoNumber true, IsIECCheckEnabled false, IsRetainMemResEnabled false, MemoryReserve 100, SetENOAutomatically false, UDAEnableTagReadback false
   VAR
      Alarm_DRP : DWord;   // Dry Run Protection Alarm
      Alarm_PS : DWord;   // Pressure Switch Alarm
   END_VAR
BEGIN

REGION Network 1: Alarm DRP
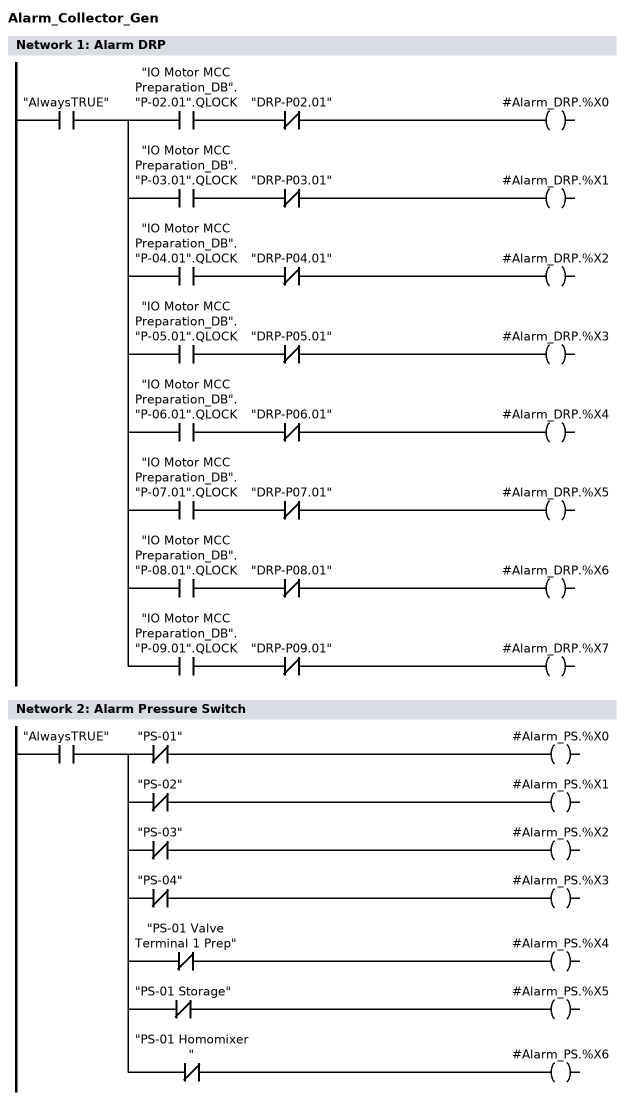
   RUNG wire#powerrail
      Contact( "AlwaysTRUE" )
      wire#w1
      Contact( "IO Motor MCC Preparation_DB"."P-02.01".QLOCK )
      I_Contact( "DRP-P02.01" )
      Coil( #Alarm_DRP.%X0 )
   END_RUNG
   RUNG wire#w1
      Contact( "IO Motor MCC Preparation_DB"."P-03.01".QLOCK )
      I_Contact( "DRP-P03.01" )
      Coil( #Alarm_DRP.%X1 )
   END_RUNG
   RUNG wire#w1
      Contact( "IO Motor MCC Preparation_DB"."P-04.01".QLOCK )
      I_Contact( "DRP-P04.01" )
      Coil( #Alarm_DRP.%X2 )
   END_RUNG
   RUNG wire#w1
      Contact( "IO Motor MCC Preparation_DB"."P-05.01".QLOCK )
      I_Contact( "DRP-P05.01" )
      Coil( #Alarm_DRP.%X3 )
   END_RUNG
   RUNG wire#w1
      Contact( "IO Motor MCC Preparation_DB"."P-06.01".QLOCK )
      I_Contact( "DRP-P06.01" )
      Coil( #Alarm_DRP.%X4 )
   END_RUNG
   RUNG wire#w1
      Contact( "IO Motor MCC Preparation_DB"."P-07.01".QLOCK )
      I_Contact( "DRP-P07.01" )
      Coil( #Alarm_DRP.%X5 )
   END_RUNG
   RUNG wire#w1
      Contact( "IO Motor MCC Preparation_DB"."P-08.01".QLOCK )
      I_Contact( "DRP-P08.01" )
      Coil( #Alarm_DRP.%X6 )
   END_RUNG
   RUNG wire#w1
      Contact( "IO Motor MCC Preparation_DB"."P-09.01".QLOCK )
      I_Contact( "DRP-P09.01" )
      Coil( #Alarm_DRP.%X7 )
   END_RUNG
   // the same network as SCL:
   #Alarm_DRP.%X0 := "AlwaysTRUE" AND "IO Motor MCC Preparation_DB"."P-02.01".QLOCK AND NOT "DRP-P02.01";
   #Alarm_DRP.%X1 := "AlwaysTRUE" AND "IO Motor MCC Preparation_DB"."P-03.01".QLOCK AND NOT "DRP-P03.01";
   #Alarm_DRP.%X2 := "AlwaysTRUE" AND "IO Motor MCC Preparation_DB"."P-04.01".QLOCK AND NOT "DRP-P04.01";
   #Alarm_DRP.%X3 := "AlwaysTRUE" AND "IO Motor MCC Preparation_DB"."P-05.01".QLOCK AND NOT "DRP-P05.01";
   #Alarm_DRP.%X4 := "AlwaysTRUE" AND "IO Motor MCC Preparation_DB"."P-06.01".QLOCK AND NOT "DRP-P06.01";
   #Alarm_DRP.%X5 := "AlwaysTRUE" AND "IO Motor MCC Preparation_DB"."P-07.01".QLOCK AND NOT "DRP-P07.01";
   #Alarm_DRP.%X6 := "AlwaysTRUE" AND "IO Motor MCC Preparation_DB"."P-08.01".QLOCK AND NOT "DRP-P08.01";
   #Alarm_DRP.%X7 := "AlwaysTRUE" AND "IO Motor MCC Preparation_DB"."P-09.01".QLOCK AND NOT "DRP-P09.01";
END_REGION

REGION Network 2: Alarm Pressure Switch
   RUNG wire#powerrail
      Contact( "AlwaysTRUE" )
      wire#w1
      I_Contact( "PS-01" )
      Coil( #Alarm_PS.%X0 )
   END_RUNG
   RUNG wire#w1
      I_Contact( "PS-02" )
      Coil( #Alarm_PS.%X1 )
   END_RUNG
   RUNG wire#w1
      I_Contact( "PS-03" )
      Coil( #Alarm_PS.%X2 )
   END_RUNG
   RUNG wire#w1
      I_Contact( "PS-04" )
      Coil( #Alarm_PS.%X3 )
   END_RUNG
   RUNG wire#w1
      I_Contact( "PS-01 Valve Terminal 1 Prep" )
      Coil( #Alarm_PS.%X4 )
   END_RUNG
   RUNG wire#w1
      I_Contact( "PS-01 Storage" )
      Coil( #Alarm_PS.%X5 )
   END_RUNG
   RUNG wire#w1
      I_Contact( "PS-01 Homomixer" )
      Coil( #Alarm_PS.%X6 )
   END_RUNG
   // the same network as SCL:
   #Alarm_PS.%X0 := "AlwaysTRUE" AND NOT "PS-01";
   #Alarm_PS.%X1 := "AlwaysTRUE" AND NOT "PS-02";
   #Alarm_PS.%X2 := "AlwaysTRUE" AND NOT "PS-03";
   #Alarm_PS.%X3 := "AlwaysTRUE" AND NOT "PS-04";
   #Alarm_PS.%X4 := "AlwaysTRUE" AND NOT "PS-01 Valve Terminal 1 Prep";
   #Alarm_PS.%X5 := "AlwaysTRUE" AND NOT "PS-01 Storage";
   #Alarm_PS.%X6 := "AlwaysTRUE" AND NOT "PS-01 Homomixer";
END_REGION
END_FUNCTION_BLOCK

FUNCTION "IO MCC Panel Blending" : Void   // FC2, LAD
{ S7_Optimized_Access := 'TRUE' }
VERSION : 0.1
// stored: AutoNumber true, IsIECCheckEnabled false, SetENOAutomatically false, UDAEnableTagReadback false
BEGIN

REGION Network 1
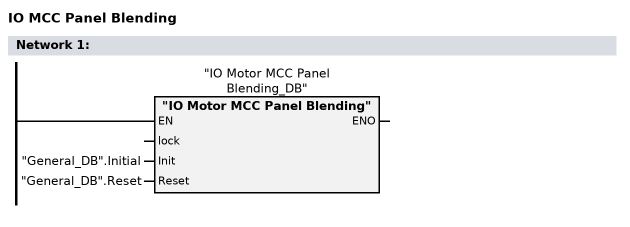
   RUNG wire#powerrail
      "IO Motor MCC Panel Blending_DB"(lock :=, Init := "General_DB".Initial, Reset := "General_DB".Reset)
   END_RUNG
   // the same network as SCL:
   "IO Motor MCC Panel Blending_DB"(Init := "General_DB".Initial, Reset := "General_DB".Reset);   // "IO Motor MCC Panel Blending"
END_REGION
END_FUNCTION

FUNCTION_BLOCK "IO Motor MCC Panel Blending"   // FB13, LAD
{ S7_Optimized_Access := 'FALSE' }
VERSION : 0.1
// stored: AutoNumber true, IsIECCheckEnabled false, SetENOAutomatically false, UDAEnableTagReadback false
   VAR_INPUT
      lock : Bool;
      Init : Bool;
      Reset : Bool;
   END_VAR
   VAR
      "XA-12.01" { S7_SetPoint := 'True'} : "Motor_w_VSD";
      "XA-13.01" { S7_SetPoint := 'True'} : "Motor_w_VSD";
      "P-13.02" { S7_SetPoint := 'True'} : "Motor";
      "XA-20.00" { S7_SetPoint := 'True'} : "Motor_w_VSD";
      "XA-21.00" { S7_SetPoint := 'True'} : "Motor_w_VSD";
      "P-21.01" { S7_SetPoint := 'True'} : "Motor_w_VSD";
      "P-22.01" { S7_SetPoint := 'True'} : "Motor_w_VSD";
      "P-22.02" { S7_SetPoint := 'True'} : "Motor";
      "P-22.03" { S7_SetPoint := 'True'} : "Motor_w_VSD";
      "P-23.01" { S7_SetPoint := 'True'} : "Motor_w_VSD";
      "P-24.01" { S7_SetPoint := 'True'} : "Motor_w_VSD";
      "P-34.01" { S7_SetPoint := 'True'} : "Motor_w_VSD";
      "XA-30.00" { S7_SetPoint := 'True'} : "Motor_w_VSD";
      "XA-31.00" { S7_SetPoint := 'True'} : "Motor_w_VSD";
      "P-31.01" { S7_SetPoint := 'True'} : "Motor_w_VSD";
      "P-32.01" { S7_SetPoint := 'True'} : "Motor_w_VSD";
      "P-32.02" { S7_SetPoint := 'True'} : "Motor";
      "P-32.03" { S7_SetPoint := 'True'} : "Motor_w_VSD";
      "P-34.02" { S7_SetPoint := 'True'} : "Motor";
      "P-35.01" { S7_SetPoint := 'True'} : "Motor_w_VSD";
      "P-22_Circ" { S7_SetPoint := 'True'} : "Motor";
      "P-32_Circ" : "Motor";
      "P-81.02" { S7_SetPoint := 'True'} : "Motor";   // CIP Return Pump Jerry Can T-81
      "P-81.01" { S7_SetPoint := 'True'} : "Motor_w_VSD";   // Transfer Pump Jerry Can T-81
      "P-34.01 DOL" { S7_SetPoint := 'True'} : "Motor_w_VSD";
      "P-84.01" { S7_SetPoint := 'True'} : "Motor_w_VSD";   // Transfer Pump Volpack Pouch T-84
      "P-84.02" { S7_SetPoint := 'True'} : "Motor_w_VSD";   // Transfer Pump Mespack DM & New T-84
      "P-82.01" { S7_SetPoint := 'True'} : "Motor_w_VSD";   // Transfer Pump Mespack P1
      "XA-14.01" { S7_SetPoint := 'True'} : "Motor_w_VSD";
      "P-20.01" { S7_SetPoint := 'True'} : "Motor_w_VSD";
      "P-30.01" { S7_SetPoint := 'True'} : "Motor_w_VSD";
      "P-40.01" { S7_SetPoint := 'True'} : "Motor_w_VSD";
      "P-41.01" { S7_SetPoint := 'True'} : "Motor_w_VSD";
      "XA-40.00" { S7_SetPoint := 'True'} : "Motor_w_VSD";
      "XA-41.00" { S7_SetPoint := 'True'} : "Motor_w_VSD";
      "P-81.02A" { S7_SetPoint := 'True'} : "Motor";   // extra fan jerry can ST-11 T-81
      "P-24.02" { S7_SetPoint := 'True'} : "Motor";   // CIP Pump Return ST 07
      "P-82.02" { S7_SetPoint := 'True'} : "Motor";   // CIP Pump Return Mespack P1 ST-16 T 85
      "XA-82.00" { S7_SetPoint := 'True'} : "Motor";   // Agitator ST-16
      "P-82.01A" { S7_SetPoint := 'True'} : "Motor";   // extra fan mespack P1 ST-16 T-85
      "P-84.01A" { S7_SetPoint := 'True'} : "Motor";   // extra fan volpack pouch ST-14 T-84
      "P-84.03" { S7_SetPoint := 'True'} : "Motor";   // CIP Pump Return Volpack Pouch ST-14 T 84
      "P-84.02A" { S7_SetPoint := 'True'} : "Motor";   // extra fan mespack new & dm ST-14 T-84
      "P-84.04" { S7_SetPoint := 'True'} : "Motor";   // CIP Pump Return Mespack New & DM ST-14 T 84
   END_VAR
   VAR_TEMP   // added for the SCL form of the ladder/FBD networks
      _w1 : Bool;
   END_VAR
BEGIN

REGION Network 1: XA-12.01 Speed
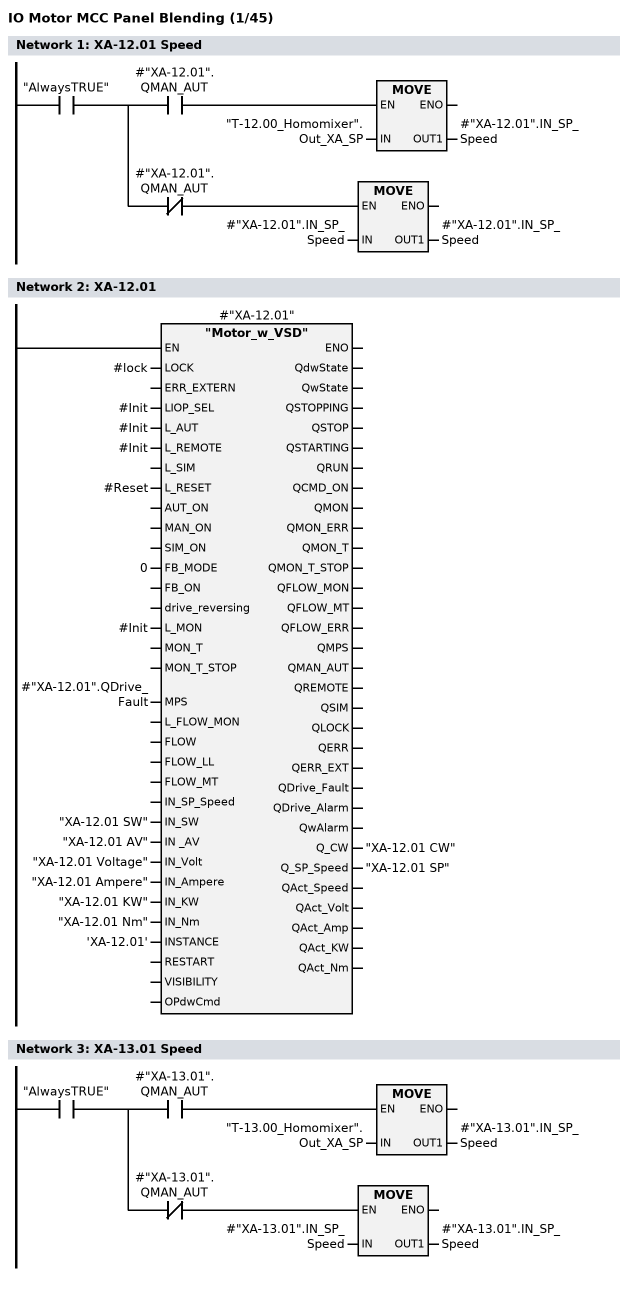
   RUNG wire#powerrail
      Contact( "AlwaysTRUE" )
      wire#w1
      Contact( #"XA-12.01".QMAN_AUT )
      Move(in := "T-12.00_Homomixer".Out_XA_SP, out1 => #"XA-12.01".IN_SP_Speed)
   END_RUNG
   RUNG wire#w1
      I_Contact( #"XA-12.01".QMAN_AUT )
      Move(in := #"XA-12.01".IN_SP_Speed, out1 => #"XA-12.01".IN_SP_Speed)
   END_RUNG
   // the same network as SCL:
   IF "AlwaysTRUE" AND #"XA-12.01".QMAN_AUT THEN
       #"XA-12.01".IN_SP_Speed := "T-12.00_Homomixer".Out_XA_SP;
   END_IF;
   IF "AlwaysTRUE" AND NOT #"XA-12.01".QMAN_AUT THEN
       #"XA-12.01".IN_SP_Speed := #"XA-12.01".IN_SP_Speed;
   END_IF;
END_REGION

REGION Network 2: XA-12.01
   RUNG wire#powerrail
      #"XA-12.01"(LOCK := #lock, ERR_EXTERN :=, LIOP_SEL := #Init, L_AUT := #Init, L_REMOTE := #Init, L_SIM :=, L_RESET := #Reset, AUT_ON :=, MAN_ON :=, SIM_ON :=, FB_MODE := 0, FB_ON :=, drive_reversing :=, L_MON := #Init, MON_T :=, MON_T_STOP :=, MPS := #"XA-12.01".QDrive_Fault, L_FLOW_MON :=, FLOW :=, FLOW_LL :=, FLOW_MT :=, IN_SP_Speed :=, IN_SW := "XA-12.01 SW", "IN _AV" := "XA-12.01 AV", IN_Volt := "XA-12.01 Voltage", IN_Ampere := "XA-12.01 Ampere", IN_KW := "XA-12.01 KW", IN_Nm := "XA-12.01 Nm", INSTANCE := 'XA-12.01', RESTART :=, VISIBILITY :=, OPdwCmd :=, QdwState =>, QwState =>, QSTOPPING =>, QSTOP =>, QSTARTING =>, QRUN =>, QCMD_ON =>, QMON =>, QMON_ERR =>, QMON_T =>, QMON_T_STOP =>, QFLOW_MON =>, QFLOW_MT =>, QFLOW_ERR =>, QMPS =>, QMAN_AUT =>, QREMOTE =>, QSIM =>, QLOCK =>, QERR =>, QERR_EXT =>, QDrive_Fault =>, QDrive_Alarm =>, QwAlarm =>, Q_CW => "XA-12.01 CW", Q_SP_Speed => "XA-12.01 SP", QAct_Speed =>, QAct_Volt =>, QAct_Amp =>, QAct_KW =>, QAct_Nm =>)
   END_RUNG
   // the same network as SCL:
   #"XA-12.01"(LOCK := #lock,   // "Motor_w_VSD"
               LIOP_SEL := #Init,
               L_AUT := #Init,
               L_REMOTE := #Init,
               L_RESET := #Reset,
               FB_MODE := 0,
               L_MON := #Init,
               MPS := #"XA-12.01".QDrive_Fault,
               IN_SW := "XA-12.01 SW",
               "IN _AV" := "XA-12.01 AV",
               IN_Volt := "XA-12.01 Voltage",
               IN_Ampere := "XA-12.01 Ampere",
               IN_KW := "XA-12.01 KW",
               IN_Nm := "XA-12.01 Nm",
               INSTANCE := 'XA-12.01',
               Q_CW => "XA-12.01 CW",
               Q_SP_Speed => "XA-12.01 SP");
END_REGION

REGION Network 3: XA-13.01 Speed
   RUNG wire#powerrail
      Contact( "AlwaysTRUE" )
      wire#w1
      Contact( #"XA-13.01".QMAN_AUT )
      Move(in := "T-13.00_Homomixer".Out_XA_SP, out1 => #"XA-13.01".IN_SP_Speed)
   END_RUNG
   RUNG wire#w1
      I_Contact( #"XA-13.01".QMAN_AUT )
      Move(in := #"XA-13.01".IN_SP_Speed, out1 => #"XA-13.01".IN_SP_Speed)
   END_RUNG
   // the same network as SCL:
   IF "AlwaysTRUE" AND #"XA-13.01".QMAN_AUT THEN
       #"XA-13.01".IN_SP_Speed := "T-13.00_Homomixer".Out_XA_SP;
   END_IF;
   IF "AlwaysTRUE" AND NOT #"XA-13.01".QMAN_AUT THEN
       #"XA-13.01".IN_SP_Speed := #"XA-13.01".IN_SP_Speed;
   END_IF;
END_REGION

REGION Network 4: XA-13.01
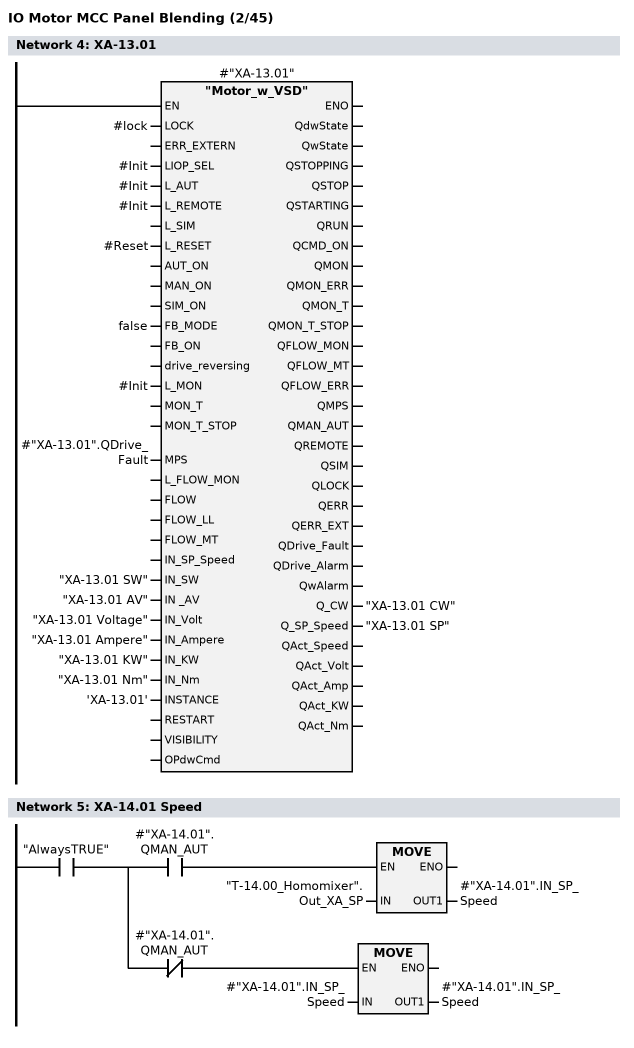
   RUNG wire#powerrail
      #"XA-13.01"(LOCK := #lock, ERR_EXTERN :=, LIOP_SEL := #Init, L_AUT := #Init, L_REMOTE := #Init, L_SIM :=, L_RESET := #Reset, AUT_ON :=, MAN_ON :=, SIM_ON :=, FB_MODE := false, FB_ON :=, drive_reversing :=, L_MON := #Init, MON_T :=, MON_T_STOP :=, MPS := #"XA-13.01".QDrive_Fault, L_FLOW_MON :=, FLOW :=, FLOW_LL :=, FLOW_MT :=, IN_SP_Speed :=, IN_SW := "XA-13.01 SW", "IN _AV" := "XA-13.01 AV", IN_Volt := "XA-13.01 Voltage", IN_Ampere := "XA-13.01 Ampere", IN_KW := "XA-13.01 KW", IN_Nm := "XA-13.01 Nm", INSTANCE := 'XA-13.01', RESTART :=, VISIBILITY :=, OPdwCmd :=, QdwState =>, QwState =>, QSTOPPING =>, QSTOP =>, QSTARTING =>, QRUN =>, QCMD_ON =>, QMON =>, QMON_ERR =>, QMON_T =>, QMON_T_STOP =>, QFLOW_MON =>, QFLOW_MT =>, QFLOW_ERR =>, QMPS =>, QMAN_AUT =>, QREMOTE =>, QSIM =>, QLOCK =>, QERR =>, QERR_EXT =>, QDrive_Fault =>, QDrive_Alarm =>, QwAlarm =>, Q_CW => "XA-13.01 CW", Q_SP_Speed => "XA-13.01 SP", QAct_Speed =>, QAct_Volt =>, QAct_Amp =>, QAct_KW =>, QAct_Nm =>)
   END_RUNG
   // the same network as SCL:
   #"XA-13.01"(LOCK := #lock,   // "Motor_w_VSD"
               LIOP_SEL := #Init,
               L_AUT := #Init,
               L_REMOTE := #Init,
               L_RESET := #Reset,
               FB_MODE := false,
               L_MON := #Init,
               MPS := #"XA-13.01".QDrive_Fault,
               IN_SW := "XA-13.01 SW",
               "IN _AV" := "XA-13.01 AV",
               IN_Volt := "XA-13.01 Voltage",
               IN_Ampere := "XA-13.01 Ampere",
               IN_KW := "XA-13.01 KW",
               IN_Nm := "XA-13.01 Nm",
               INSTANCE := 'XA-13.01',
               Q_CW => "XA-13.01 CW",
               Q_SP_Speed => "XA-13.01 SP");
END_REGION

REGION Network 5: XA-14.01 Speed
   RUNG wire#powerrail
      Contact( "AlwaysTRUE" )
      wire#w1
      Contact( #"XA-14.01".QMAN_AUT )
      Move(in := "T-14.00_Homomixer".Out_XA_SP, out1 => #"XA-14.01".IN_SP_Speed)
   END_RUNG
   RUNG wire#w1
      I_Contact( #"XA-14.01".QMAN_AUT )
      Move(in := #"XA-14.01".IN_SP_Speed, out1 => #"XA-14.01".IN_SP_Speed)
   END_RUNG
   // the same network as SCL:
   IF "AlwaysTRUE" AND #"XA-14.01".QMAN_AUT THEN
       #"XA-14.01".IN_SP_Speed := "T-14.00_Homomixer".Out_XA_SP;
   END_IF;
   IF "AlwaysTRUE" AND NOT #"XA-14.01".QMAN_AUT THEN
       #"XA-14.01".IN_SP_Speed := #"XA-14.01".IN_SP_Speed;
   END_IF;
END_REGION

REGION Network 6: XA-14.01
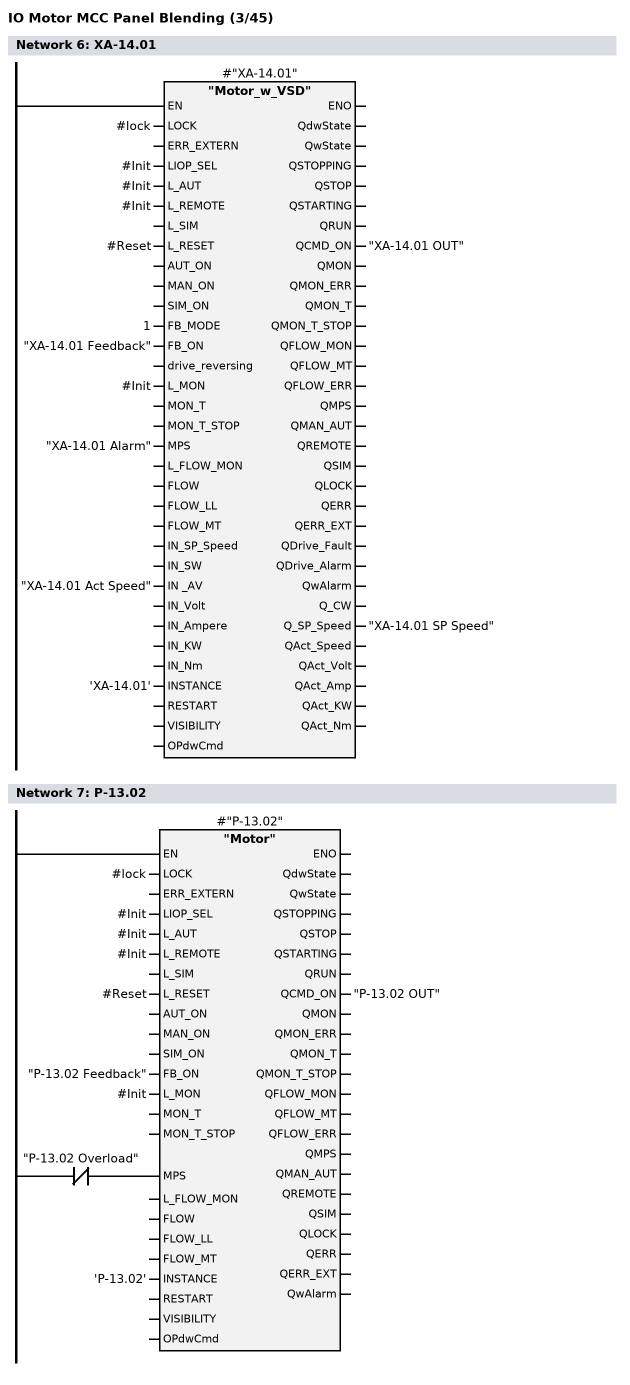
   RUNG wire#powerrail
      #"XA-14.01"(LOCK := #lock, ERR_EXTERN :=, LIOP_SEL := #Init, L_AUT := #Init, L_REMOTE := #Init, L_SIM :=, L_RESET := #Reset, AUT_ON :=, MAN_ON :=, SIM_ON :=, FB_MODE := 1, FB_ON := "XA-14.01 Feedback", drive_reversing :=, L_MON := #Init, MON_T :=, MON_T_STOP :=, MPS := "XA-14.01 Alarm", L_FLOW_MON :=, FLOW :=, FLOW_LL :=, FLOW_MT :=, IN_SP_Speed :=, IN_SW :=, "IN _AV" := "XA-14.01 Act Speed", IN_Volt :=, IN_Ampere :=, IN_KW :=, IN_Nm :=, INSTANCE := 'XA-14.01', RESTART :=, VISIBILITY :=, OPdwCmd :=, QdwState =>, QwState =>, QSTOPPING =>, QSTOP =>, QSTARTING =>, QRUN =>, QCMD_ON => "XA-14.01 OUT", QMON =>, QMON_ERR =>, QMON_T =>, QMON_T_STOP =>, QFLOW_MON =>, QFLOW_MT =>, QFLOW_ERR =>, QMPS =>, QMAN_AUT =>, QREMOTE =>, QSIM =>, QLOCK =>, QERR =>, QERR_EXT =>, QDrive_Fault =>, QDrive_Alarm =>, QwAlarm =>, Q_CW =>, Q_SP_Speed => "XA-14.01 SP Speed", QAct_Speed =>, QAct_Volt =>, QAct_Amp =>, QAct_KW =>, QAct_Nm =>)
   END_RUNG
   // the same network as SCL:
   #"XA-14.01"(LOCK := #lock,   // "Motor_w_VSD"
               LIOP_SEL := #Init,
               L_AUT := #Init,
               L_REMOTE := #Init,
               L_RESET := #Reset,
               FB_MODE := 1,
               FB_ON := "XA-14.01 Feedback",
               L_MON := #Init,
               MPS := "XA-14.01 Alarm",
               "IN _AV" := "XA-14.01 Act Speed",
               INSTANCE := 'XA-14.01',
               QCMD_ON => "XA-14.01 OUT",
               Q_SP_Speed => "XA-14.01 SP Speed");
END_REGION

REGION Network 7: P-13.02
   RUNG wire#powerrail
      #"P-13.02"(MPS := wire#w1, LOCK := #lock, ERR_EXTERN :=, LIOP_SEL := #Init, L_AUT := #Init, L_REMOTE := #Init, L_SIM :=, L_RESET := #Reset, AUT_ON :=, MAN_ON :=, SIM_ON :=, FB_ON := "P-13.02 Feedback", L_MON := #Init, MON_T :=, MON_T_STOP :=, L_FLOW_MON :=, FLOW :=, FLOW_LL :=, FLOW_MT :=, INSTANCE := 'P-13.02', RESTART :=, VISIBILITY :=, OPdwCmd :=, QdwState =>, QwState =>, QSTOPPING =>, QSTOP =>, QSTARTING =>, QRUN =>, QCMD_ON => "P-13.02 OUT", QMON =>, QMON_ERR =>, QMON_T =>, QMON_T_STOP =>, QFLOW_MON =>, QFLOW_MT =>, QFLOW_ERR =>, QMPS =>, QMAN_AUT =>, QREMOTE =>, QSIM =>, QLOCK =>, QERR =>, QERR_EXT =>, QwAlarm =>)
   END_RUNG
   RUNG wire#powerrail
      I_Contact( "P-13.02 Overload" )
   END_RUNG wire#w1
   // the same network as SCL:
   #"P-13.02"(LOCK := #lock,   // "Motor"
              LIOP_SEL := #Init,
              L_AUT := #Init,
              L_REMOTE := #Init,
              L_RESET := #Reset,
              FB_ON := "P-13.02 Feedback",
              L_MON := #Init,
              MPS := NOT "P-13.02 Overload",
              INSTANCE := 'P-13.02',
              QCMD_ON => "P-13.02 OUT");
END_REGION

REGION Network 9: XA-20.00 Speed
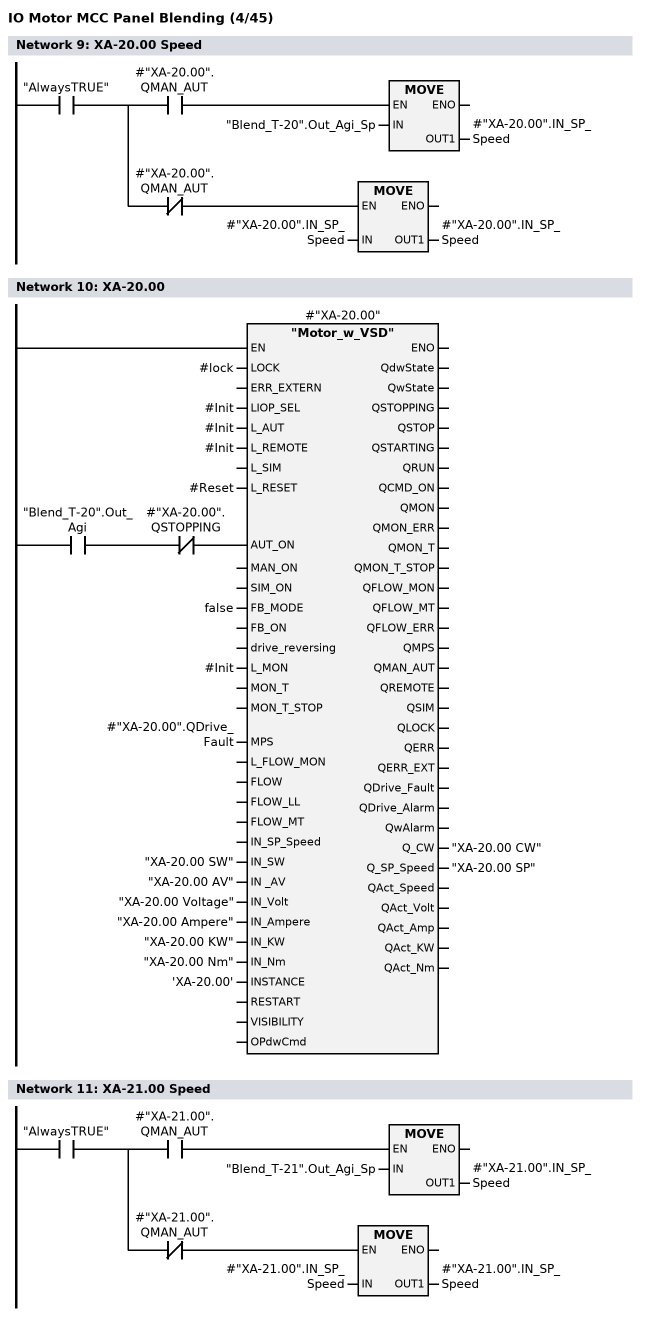
   RUNG wire#powerrail
      Contact( "AlwaysTRUE" )
      wire#w1
      Contact( #"XA-20.00".QMAN_AUT )
      Move(in := "Blend_T-20".Out_Agi_Sp, out1 => #"XA-20.00".IN_SP_Speed)
   END_RUNG
   RUNG wire#w1
      I_Contact( #"XA-20.00".QMAN_AUT )
      Move(in := #"XA-20.00".IN_SP_Speed, out1 => #"XA-20.00".IN_SP_Speed)
   END_RUNG
   // the same network as SCL:
   IF "AlwaysTRUE" AND #"XA-20.00".QMAN_AUT THEN #"XA-20.00".IN_SP_Speed := "Blend_T-20".Out_Agi_Sp; END_IF;
   IF "AlwaysTRUE" AND NOT #"XA-20.00".QMAN_AUT THEN
       #"XA-20.00".IN_SP_Speed := #"XA-20.00".IN_SP_Speed;
   END_IF;
END_REGION

REGION Network 10: XA-20.00
   RUNG wire#powerrail
      #"XA-20.00"(AUT_ON := wire#w1, LOCK := #lock, ERR_EXTERN :=, LIOP_SEL := #Init, L_AUT := #Init, L_REMOTE := #Init, L_SIM :=, L_RESET := #Reset, MAN_ON :=, SIM_ON :=, FB_MODE := false, FB_ON :=, drive_reversing :=, L_MON := #Init, MON_T :=, MON_T_STOP :=, MPS := #"XA-20.00".QDrive_Fault, L_FLOW_MON :=, FLOW :=, FLOW_LL :=, FLOW_MT :=, IN_SP_Speed :=, IN_SW := "XA-20.00 SW", "IN _AV" := "XA-20.00 AV", IN_Volt := "XA-20.00 Voltage", IN_Ampere := "XA-20.00 Ampere", IN_KW := "XA-20.00 KW", IN_Nm := "XA-20.00 Nm", INSTANCE := 'XA-20.00', RESTART :=, VISIBILITY :=, OPdwCmd :=, QdwState =>, QwState =>, QSTOPPING =>, QSTOP =>, QSTARTING =>, QRUN =>, QCMD_ON =>, QMON =>, QMON_ERR =>, QMON_T =>, QMON_T_STOP =>, QFLOW_MON =>, QFLOW_MT =>, QFLOW_ERR =>, QMPS =>, QMAN_AUT =>, QREMOTE =>, QSIM =>, QLOCK =>, QERR =>, QERR_EXT =>, QDrive_Fault =>, QDrive_Alarm =>, QwAlarm =>, Q_CW => "XA-20.00 CW", Q_SP_Speed => "XA-20.00 SP", QAct_Speed =>, QAct_Volt =>, QAct_Amp =>, QAct_KW =>, QAct_Nm =>)
   END_RUNG
   RUNG wire#powerrail
      Contact( "Blend_T-20".Out_Agi )
      I_Contact( #"XA-20.00".QSTOPPING )
   END_RUNG wire#w1
   // the same network as SCL:
   #"XA-20.00"(LOCK := #lock,   // "Motor_w_VSD"
               LIOP_SEL := #Init,
               L_AUT := #Init,
               L_REMOTE := #Init,
               L_RESET := #Reset,
               AUT_ON := "Blend_T-20".Out_Agi AND NOT #"XA-20.00".QSTOPPING,
               FB_MODE := false,
               L_MON := #Init,
               MPS := #"XA-20.00".QDrive_Fault,
               IN_SW := "XA-20.00 SW",
               "IN _AV" := "XA-20.00 AV",
               IN_Volt := "XA-20.00 Voltage",
               IN_Ampere := "XA-20.00 Ampere",
               IN_KW := "XA-20.00 KW",
               IN_Nm := "XA-20.00 Nm",
               INSTANCE := 'XA-20.00',
               Q_CW => "XA-20.00 CW",
               Q_SP_Speed => "XA-20.00 SP");
END_REGION

REGION Network 11: XA-21.00 Speed
   RUNG wire#powerrail
      Contact( "AlwaysTRUE" )
      wire#w1
      Contact( #"XA-21.00".QMAN_AUT )
      Move(in := "Blend_T-21".Out_Agi_Sp, out1 => #"XA-21.00".IN_SP_Speed)
   END_RUNG
   RUNG wire#w1
      I_Contact( #"XA-21.00".QMAN_AUT )
      Move(in := #"XA-21.00".IN_SP_Speed, out1 => #"XA-21.00".IN_SP_Speed)
   END_RUNG
   // the same network as SCL:
   IF "AlwaysTRUE" AND #"XA-21.00".QMAN_AUT THEN #"XA-21.00".IN_SP_Speed := "Blend_T-21".Out_Agi_Sp; END_IF;
   IF "AlwaysTRUE" AND NOT #"XA-21.00".QMAN_AUT THEN
       #"XA-21.00".IN_SP_Speed := #"XA-21.00".IN_SP_Speed;
   END_IF;
END_REGION

REGION Network 12: XA-21.00
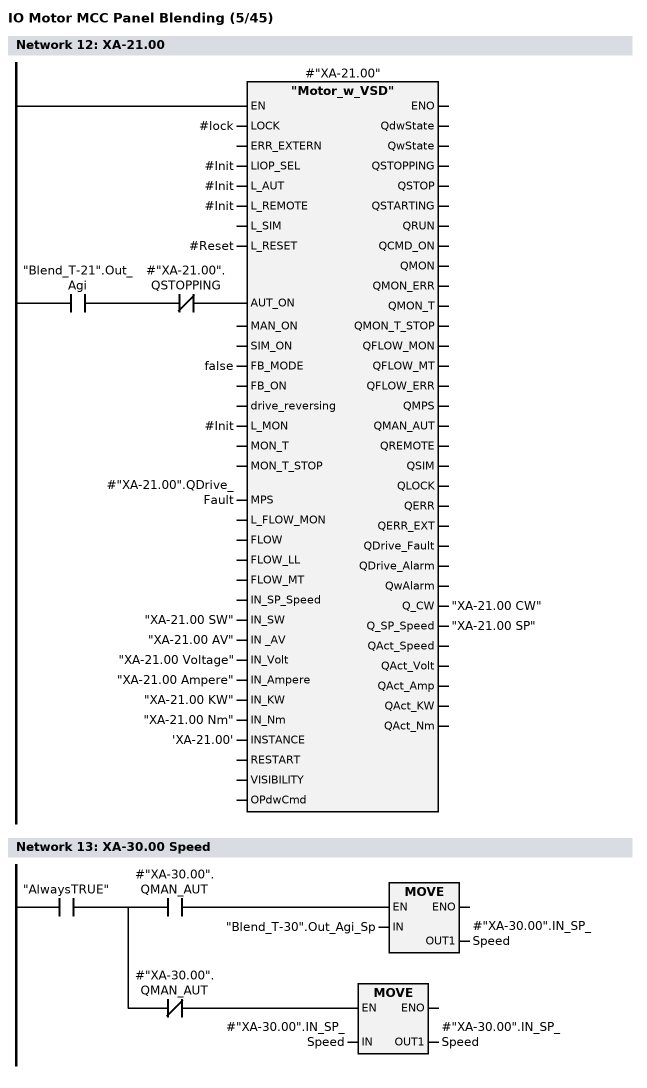
   RUNG wire#powerrail
      #"XA-21.00"(AUT_ON := wire#w1, LOCK := #lock, ERR_EXTERN :=, LIOP_SEL := #Init, L_AUT := #Init, L_REMOTE := #Init, L_SIM :=, L_RESET := #Reset, MAN_ON :=, SIM_ON :=, FB_MODE := false, FB_ON :=, drive_reversing :=, L_MON := #Init, MON_T :=, MON_T_STOP :=, MPS := #"XA-21.00".QDrive_Fault, L_FLOW_MON :=, FLOW :=, FLOW_LL :=, FLOW_MT :=, IN_SP_Speed :=, IN_SW := "XA-21.00 SW", "IN _AV" := "XA-21.00 AV", IN_Volt := "XA-21.00 Voltage", IN_Ampere := "XA-21.00 Ampere", IN_KW := "XA-21.00 KW", IN_Nm := "XA-21.00 Nm", INSTANCE := 'XA-21.00', RESTART :=, VISIBILITY :=, OPdwCmd :=, QdwState =>, QwState =>, QSTOPPING =>, QSTOP =>, QSTARTING =>, QRUN =>, QCMD_ON =>, QMON =>, QMON_ERR =>, QMON_T =>, QMON_T_STOP =>, QFLOW_MON =>, QFLOW_MT =>, QFLOW_ERR =>, QMPS =>, QMAN_AUT =>, QREMOTE =>, QSIM =>, QLOCK =>, QERR =>, QERR_EXT =>, QDrive_Fault =>, QDrive_Alarm =>, QwAlarm =>, Q_CW => "XA-21.00 CW", Q_SP_Speed => "XA-21.00 SP", QAct_Speed =>, QAct_Volt =>, QAct_Amp =>, QAct_KW =>, QAct_Nm =>)
   END_RUNG
   RUNG wire#powerrail
      Contact( "Blend_T-21".Out_Agi )
      I_Contact( #"XA-21.00".QSTOPPING )
   END_RUNG wire#w1
   // the same network as SCL:
   #"XA-21.00"(LOCK := #lock,   // "Motor_w_VSD"
               LIOP_SEL := #Init,
               L_AUT := #Init,
               L_REMOTE := #Init,
               L_RESET := #Reset,
               AUT_ON := "Blend_T-21".Out_Agi AND NOT #"XA-21.00".QSTOPPING,
               FB_MODE := false,
               L_MON := #Init,
               MPS := #"XA-21.00".QDrive_Fault,
               IN_SW := "XA-21.00 SW",
               "IN _AV" := "XA-21.00 AV",
               IN_Volt := "XA-21.00 Voltage",
               IN_Ampere := "XA-21.00 Ampere",
               IN_KW := "XA-21.00 KW",
               IN_Nm := "XA-21.00 Nm",
               INSTANCE := 'XA-21.00',
               Q_CW => "XA-21.00 CW",
               Q_SP_Speed => "XA-21.00 SP");
END_REGION

REGION Network 13: XA-30.00 Speed
   RUNG wire#powerrail
      Contact( "AlwaysTRUE" )
      wire#w1
      Contact( #"XA-30.00".QMAN_AUT )
      Move(in := "Blend_T-30".Out_Agi_Sp, out1 => #"XA-30.00".IN_SP_Speed)
   END_RUNG
   RUNG wire#w1
      I_Contact( #"XA-30.00".QMAN_AUT )
      Move(in := #"XA-30.00".IN_SP_Speed, out1 => #"XA-30.00".IN_SP_Speed)
   END_RUNG
   // the same network as SCL:
   IF "AlwaysTRUE" AND #"XA-30.00".QMAN_AUT THEN #"XA-30.00".IN_SP_Speed := "Blend_T-30".Out_Agi_Sp; END_IF;
   IF "AlwaysTRUE" AND NOT #"XA-30.00".QMAN_AUT THEN
       #"XA-30.00".IN_SP_Speed := #"XA-30.00".IN_SP_Speed;
   END_IF;
END_REGION

REGION Network 14: XA-30.00
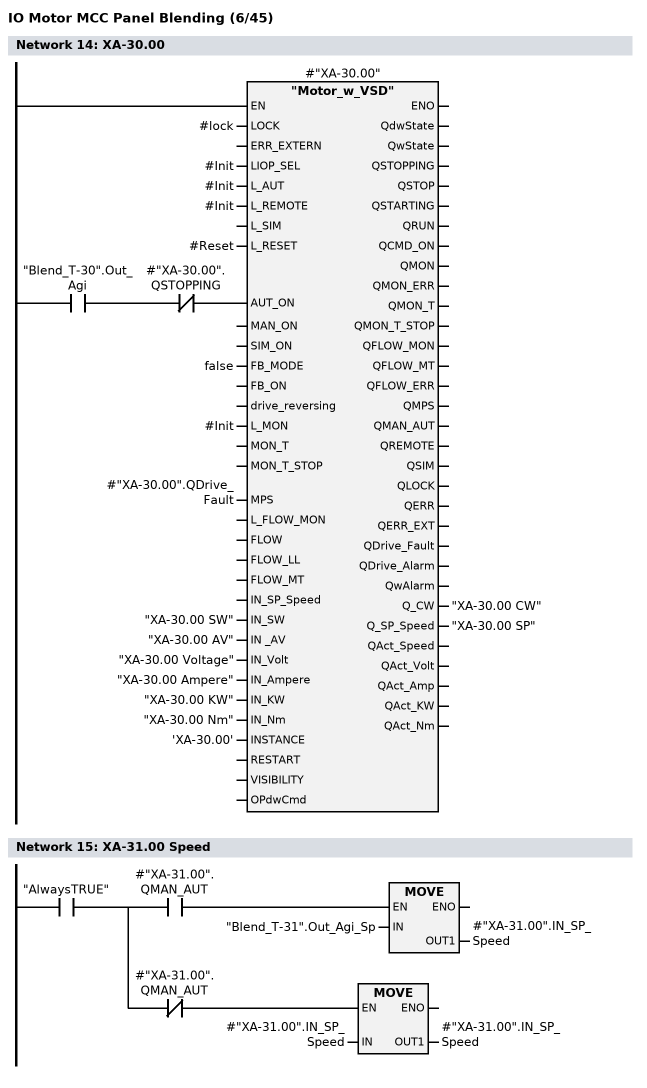
   RUNG wire#powerrail
      #"XA-30.00"(AUT_ON := wire#w1, LOCK := #lock, ERR_EXTERN :=, LIOP_SEL := #Init, L_AUT := #Init, L_REMOTE := #Init, L_SIM :=, L_RESET := #Reset, MAN_ON :=, SIM_ON :=, FB_MODE := false, FB_ON :=, drive_reversing :=, L_MON := #Init, MON_T :=, MON_T_STOP :=, MPS := #"XA-30.00".QDrive_Fault, L_FLOW_MON :=, FLOW :=, FLOW_LL :=, FLOW_MT :=, IN_SP_Speed :=, IN_SW := "XA-30.00 SW", "IN _AV" := "XA-30.00 AV", IN_Volt := "XA-30.00 Voltage", IN_Ampere := "XA-30.00 Ampere", IN_KW := "XA-30.00 KW", IN_Nm := "XA-30.00 Nm", INSTANCE := 'XA-30.00', RESTART :=, VISIBILITY :=, OPdwCmd :=, QdwState =>, QwState =>, QSTOPPING =>, QSTOP =>, QSTARTING =>, QRUN =>, QCMD_ON =>, QMON =>, QMON_ERR =>, QMON_T =>, QMON_T_STOP =>, QFLOW_MON =>, QFLOW_MT =>, QFLOW_ERR =>, QMPS =>, QMAN_AUT =>, QREMOTE =>, QSIM =>, QLOCK =>, QERR =>, QERR_EXT =>, QDrive_Fault =>, QDrive_Alarm =>, QwAlarm =>, Q_CW => "XA-30.00 CW", Q_SP_Speed => "XA-30.00 SP", QAct_Speed =>, QAct_Volt =>, QAct_Amp =>, QAct_KW =>, QAct_Nm =>)
   END_RUNG
   RUNG wire#powerrail
      Contact( "Blend_T-30".Out_Agi )
      I_Contact( #"XA-30.00".QSTOPPING )
   END_RUNG wire#w1
   // the same network as SCL:
   #"XA-30.00"(LOCK := #lock,   // "Motor_w_VSD"
               LIOP_SEL := #Init,
               L_AUT := #Init,
               L_REMOTE := #Init,
               L_RESET := #Reset,
               AUT_ON := "Blend_T-30".Out_Agi AND NOT #"XA-30.00".QSTOPPING,
               FB_MODE := false,
               L_MON := #Init,
               MPS := #"XA-30.00".QDrive_Fault,
               IN_SW := "XA-30.00 SW",
               "IN _AV" := "XA-30.00 AV",
               IN_Volt := "XA-30.00 Voltage",
               IN_Ampere := "XA-30.00 Ampere",
               IN_KW := "XA-30.00 KW",
               IN_Nm := "XA-30.00 Nm",
               INSTANCE := 'XA-30.00',
               Q_CW => "XA-30.00 CW",
               Q_SP_Speed => "XA-30.00 SP");
END_REGION

REGION Network 15: XA-31.00 Speed
   RUNG wire#powerrail
      Contact( "AlwaysTRUE" )
      wire#w1
      Contact( #"XA-31.00".QMAN_AUT )
      Move(in := "Blend_T-31".Out_Agi_Sp, out1 => #"XA-31.00".IN_SP_Speed)
   END_RUNG
   RUNG wire#w1
      I_Contact( #"XA-31.00".QMAN_AUT )
      Move(in := #"XA-31.00".IN_SP_Speed, out1 => #"XA-31.00".IN_SP_Speed)
   END_RUNG
   // the same network as SCL:
   IF "AlwaysTRUE" AND #"XA-31.00".QMAN_AUT THEN #"XA-31.00".IN_SP_Speed := "Blend_T-31".Out_Agi_Sp; END_IF;
   IF "AlwaysTRUE" AND NOT #"XA-31.00".QMAN_AUT THEN
       #"XA-31.00".IN_SP_Speed := #"XA-31.00".IN_SP_Speed;
   END_IF;
END_REGION

REGION Network 16: XA-31.00
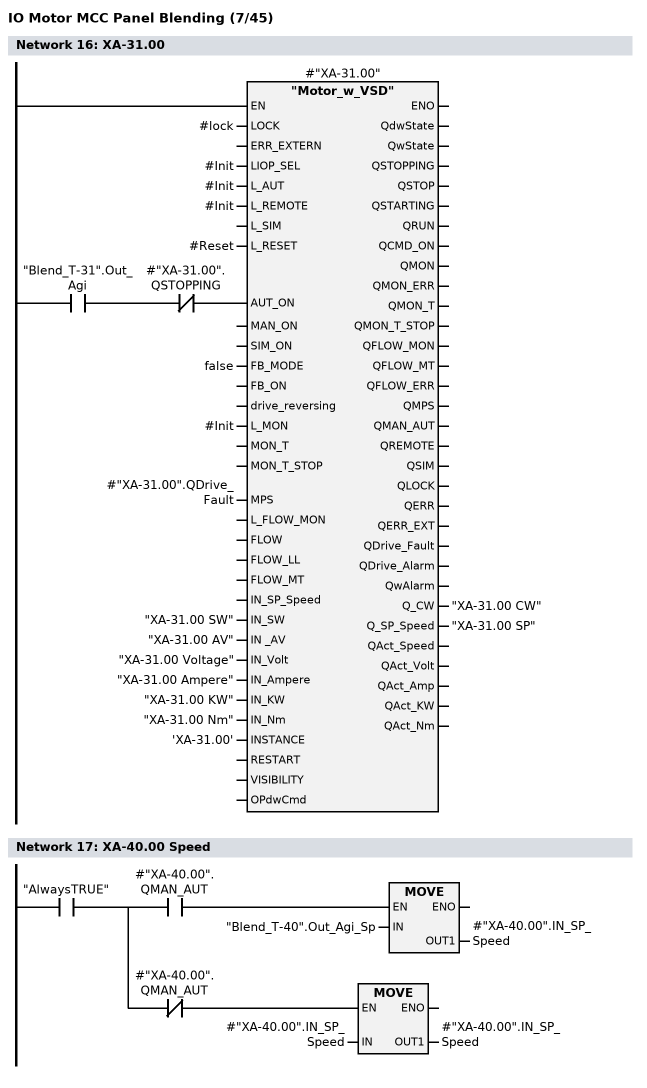
   RUNG wire#powerrail
      #"XA-31.00"(AUT_ON := wire#w1, LOCK := #lock, ERR_EXTERN :=, LIOP_SEL := #Init, L_AUT := #Init, L_REMOTE := #Init, L_SIM :=, L_RESET := #Reset, MAN_ON :=, SIM_ON :=, FB_MODE := false, FB_ON :=, drive_reversing :=, L_MON := #Init, MON_T :=, MON_T_STOP :=, MPS := #"XA-31.00".QDrive_Fault, L_FLOW_MON :=, FLOW :=, FLOW_LL :=, FLOW_MT :=, IN_SP_Speed :=, IN_SW := "XA-31.00 SW", "IN _AV" := "XA-31.00 AV", IN_Volt := "XA-31.00 Voltage", IN_Ampere := "XA-31.00 Ampere", IN_KW := "XA-31.00 KW", IN_Nm := "XA-31.00 Nm", INSTANCE := 'XA-31.00', RESTART :=, VISIBILITY :=, OPdwCmd :=, QdwState =>, QwState =>, QSTOPPING =>, QSTOP =>, QSTARTING =>, QRUN =>, QCMD_ON =>, QMON =>, QMON_ERR =>, QMON_T =>, QMON_T_STOP =>, QFLOW_MON =>, QFLOW_MT =>, QFLOW_ERR =>, QMPS =>, QMAN_AUT =>, QREMOTE =>, QSIM =>, QLOCK =>, QERR =>, QERR_EXT =>, QDrive_Fault =>, QDrive_Alarm =>, QwAlarm =>, Q_CW => "XA-31.00 CW", Q_SP_Speed => "XA-31.00 SP", QAct_Speed =>, QAct_Volt =>, QAct_Amp =>, QAct_KW =>, QAct_Nm =>)
   END_RUNG
   RUNG wire#powerrail
      Contact( "Blend_T-31".Out_Agi )
      I_Contact( #"XA-31.00".QSTOPPING )
   END_RUNG wire#w1
   // the same network as SCL:
   #"XA-31.00"(LOCK := #lock,   // "Motor_w_VSD"
               LIOP_SEL := #Init,
               L_AUT := #Init,
               L_REMOTE := #Init,
               L_RESET := #Reset,
               AUT_ON := "Blend_T-31".Out_Agi AND NOT #"XA-31.00".QSTOPPING,
               FB_MODE := false,
               L_MON := #Init,
               MPS := #"XA-31.00".QDrive_Fault,
               IN_SW := "XA-31.00 SW",
               "IN _AV" := "XA-31.00 AV",
               IN_Volt := "XA-31.00 Voltage",
               IN_Ampere := "XA-31.00 Ampere",
               IN_KW := "XA-31.00 KW",
               IN_Nm := "XA-31.00 Nm",
               INSTANCE := 'XA-31.00',
               Q_CW => "XA-31.00 CW",
               Q_SP_Speed => "XA-31.00 SP");
END_REGION

REGION Network 17: XA-40.00 Speed
   RUNG wire#powerrail
      Contact( "AlwaysTRUE" )
      wire#w1
      Contact( #"XA-40.00".QMAN_AUT )
      Move(in := "Blend_T-40".Out_Agi_Sp, out1 => #"XA-40.00".IN_SP_Speed)
   END_RUNG
   RUNG wire#w1
      I_Contact( #"XA-40.00".QMAN_AUT )
      Move(in := #"XA-40.00".IN_SP_Speed, out1 => #"XA-40.00".IN_SP_Speed)
   END_RUNG
   // the same network as SCL:
   IF "AlwaysTRUE" AND #"XA-40.00".QMAN_AUT THEN #"XA-40.00".IN_SP_Speed := "Blend_T-40".Out_Agi_Sp; END_IF;
   IF "AlwaysTRUE" AND NOT #"XA-40.00".QMAN_AUT THEN
       #"XA-40.00".IN_SP_Speed := #"XA-40.00".IN_SP_Speed;
   END_IF;
END_REGION

REGION Network 18: XA-40.00
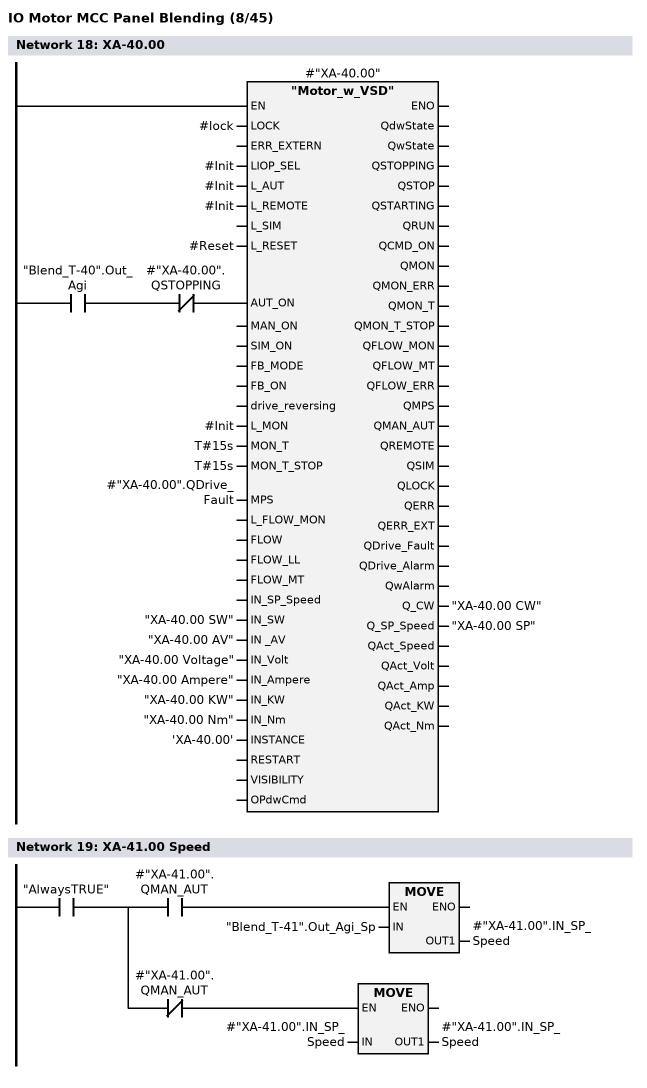
   RUNG wire#powerrail
      #"XA-40.00"(AUT_ON := wire#w1, LOCK := #lock, ERR_EXTERN :=, LIOP_SEL := #Init, L_AUT := #Init, L_REMOTE := #Init, L_SIM :=, L_RESET := #Reset, MAN_ON :=, SIM_ON :=, FB_MODE :=, FB_ON :=, drive_reversing :=, L_MON := #Init, MON_T := T#15s, MON_T_STOP := T#15s, MPS := #"XA-40.00".QDrive_Fault, L_FLOW_MON :=, FLOW :=, FLOW_LL :=, FLOW_MT :=, IN_SP_Speed :=, IN_SW := "XA-40.00 SW", "IN _AV" := "XA-40.00 AV", IN_Volt := "XA-40.00 Voltage", IN_Ampere := "XA-40.00 Ampere", IN_KW := "XA-40.00 KW", IN_Nm := "XA-40.00 Nm", INSTANCE := 'XA-40.00', RESTART :=, VISIBILITY :=, OPdwCmd :=, QdwState =>, QwState =>, QSTOPPING =>, QSTOP =>, QSTARTING =>, QRUN =>, QCMD_ON =>, QMON =>, QMON_ERR =>, QMON_T =>, QMON_T_STOP =>, QFLOW_MON =>, QFLOW_MT =>, QFLOW_ERR =>, QMPS =>, QMAN_AUT =>, QREMOTE =>, QSIM =>, QLOCK =>, QERR =>, QERR_EXT =>, QDrive_Fault =>, QDrive_Alarm =>, QwAlarm =>, Q_CW => "XA-40.00 CW", Q_SP_Speed => "XA-40.00 SP", QAct_Speed =>, QAct_Volt =>, QAct_Amp =>, QAct_KW =>, QAct_Nm =>)
   END_RUNG
   RUNG wire#powerrail
      Contact( "Blend_T-40".Out_Agi )
      I_Contact( #"XA-40.00".QSTOPPING )
   END_RUNG wire#w1
   // the same network as SCL:
   #"XA-40.00"(LOCK := #lock,   // "Motor_w_VSD"
               LIOP_SEL := #Init,
               L_AUT := #Init,
               L_REMOTE := #Init,
               L_RESET := #Reset,
               AUT_ON := "Blend_T-40".Out_Agi AND NOT #"XA-40.00".QSTOPPING,
               L_MON := #Init,
               MON_T := T#15s,
               MON_T_STOP := T#15s,
               MPS := #"XA-40.00".QDrive_Fault,
               IN_SW := "XA-40.00 SW",
               "IN _AV" := "XA-40.00 AV",
               IN_Volt := "XA-40.00 Voltage",
               IN_Ampere := "XA-40.00 Ampere",
               IN_KW := "XA-40.00 KW",
               IN_Nm := "XA-40.00 Nm",
               INSTANCE := 'XA-40.00',
               Q_CW => "XA-40.00 CW",
               Q_SP_Speed => "XA-40.00 SP");
END_REGION

REGION Network 19: XA-41.00 Speed
   RUNG wire#powerrail
      Contact( "AlwaysTRUE" )
      wire#w1
      Contact( #"XA-41.00".QMAN_AUT )
      Move(in := "Blend_T-41".Out_Agi_Sp, out1 => #"XA-41.00".IN_SP_Speed)
   END_RUNG
   RUNG wire#w1
      I_Contact( #"XA-41.00".QMAN_AUT )
      Move(in := #"XA-41.00".IN_SP_Speed, out1 => #"XA-41.00".IN_SP_Speed)
   END_RUNG
   // the same network as SCL:
   IF "AlwaysTRUE" AND #"XA-41.00".QMAN_AUT THEN #"XA-41.00".IN_SP_Speed := "Blend_T-41".Out_Agi_Sp; END_IF;
   IF "AlwaysTRUE" AND NOT #"XA-41.00".QMAN_AUT THEN
       #"XA-41.00".IN_SP_Speed := #"XA-41.00".IN_SP_Speed;
   END_IF;
END_REGION

REGION Network 20: XA-41.00
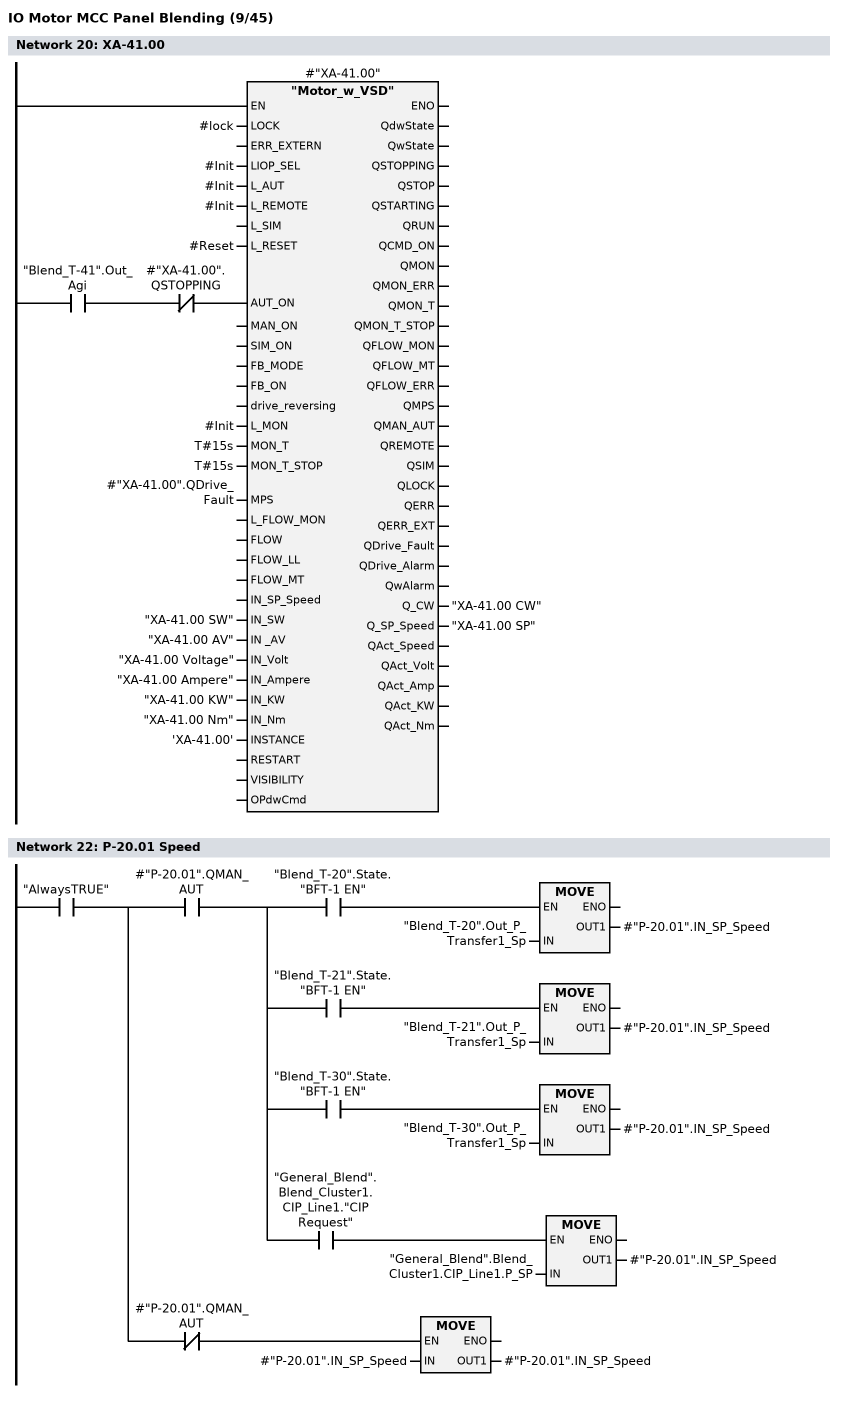
   RUNG wire#powerrail
      #"XA-41.00"(AUT_ON := wire#w1, LOCK := #lock, ERR_EXTERN :=, LIOP_SEL := #Init, L_AUT := #Init, L_REMOTE := #Init, L_SIM :=, L_RESET := #Reset, MAN_ON :=, SIM_ON :=, FB_MODE :=, FB_ON :=, drive_reversing :=, L_MON := #Init, MON_T := T#15s, MON_T_STOP := T#15s, MPS := #"XA-41.00".QDrive_Fault, L_FLOW_MON :=, FLOW :=, FLOW_LL :=, FLOW_MT :=, IN_SP_Speed :=, IN_SW := "XA-41.00 SW", "IN _AV" := "XA-41.00 AV", IN_Volt := "XA-41.00 Voltage", IN_Ampere := "XA-41.00 Ampere", IN_KW := "XA-41.00 KW", IN_Nm := "XA-41.00 Nm", INSTANCE := 'XA-41.00', RESTART :=, VISIBILITY :=, OPdwCmd :=, QdwState =>, QwState =>, QSTOPPING =>, QSTOP =>, QSTARTING =>, QRUN =>, QCMD_ON =>, QMON =>, QMON_ERR =>, QMON_T =>, QMON_T_STOP =>, QFLOW_MON =>, QFLOW_MT =>, QFLOW_ERR =>, QMPS =>, QMAN_AUT =>, QREMOTE =>, QSIM =>, QLOCK =>, QERR =>, QERR_EXT =>, QDrive_Fault =>, QDrive_Alarm =>, QwAlarm =>, Q_CW => "XA-41.00 CW", Q_SP_Speed => "XA-41.00 SP", QAct_Speed =>, QAct_Volt =>, QAct_Amp =>, QAct_KW =>, QAct_Nm =>)
   END_RUNG
   RUNG wire#powerrail
      Contact( "Blend_T-41".Out_Agi )
      I_Contact( #"XA-41.00".QSTOPPING )
   END_RUNG wire#w1
   // the same network as SCL:
   #"XA-41.00"(LOCK := #lock,   // "Motor_w_VSD"
               LIOP_SEL := #Init,
               L_AUT := #Init,
               L_REMOTE := #Init,
               L_RESET := #Reset,
               AUT_ON := "Blend_T-41".Out_Agi AND NOT #"XA-41.00".QSTOPPING,
               L_MON := #Init,
               MON_T := T#15s,
               MON_T_STOP := T#15s,
               MPS := #"XA-41.00".QDrive_Fault,
               IN_SW := "XA-41.00 SW",
               "IN _AV" := "XA-41.00 AV",
               IN_Volt := "XA-41.00 Voltage",
               IN_Ampere := "XA-41.00 Ampere",
               IN_KW := "XA-41.00 KW",
               IN_Nm := "XA-41.00 Nm",
               INSTANCE := 'XA-41.00',
               Q_CW => "XA-41.00 CW",
               Q_SP_Speed => "XA-41.00 SP");
END_REGION

REGION Network 22: P-20.01 Speed
   RUNG wire#powerrail
      Contact( "AlwaysTRUE" )
      wire#w1
      Contact( #"P-20.01".QMAN_AUT )
      wire#w2
      Contact( "Blend_T-20".State."BFT-1 EN" )
      Move(in := "Blend_T-20".Out_P_Transfer1_Sp, out1 => #"P-20.01".IN_SP_Speed)
   END_RUNG
   RUNG wire#w2
      Contact( "Blend_T-21".State."BFT-1 EN" )
      Move(in := "Blend_T-21".Out_P_Transfer1_Sp, out1 => #"P-20.01".IN_SP_Speed)
   END_RUNG
   RUNG wire#w2
      Contact( "Blend_T-30".State."BFT-1 EN" )
      Move(in := "Blend_T-30".Out_P_Transfer1_Sp, out1 => #"P-20.01".IN_SP_Speed)
   END_RUNG
   RUNG wire#w2
      Contact( "General_Blend".Blend_Cluster1.CIP_Line1."CIP Request" )
      Move(in := "General_Blend".Blend_Cluster1.CIP_Line1.P_SP, out1 => #"P-20.01".IN_SP_Speed)
   END_RUNG
   RUNG wire#w1
      I_Contact( #"P-20.01".QMAN_AUT )
      Move(in := #"P-20.01".IN_SP_Speed, out1 => #"P-20.01".IN_SP_Speed)
   END_RUNG
   // the same network as SCL:
   #_w1 := "AlwaysTRUE" AND #"P-20.01".QMAN_AUT;
   IF #_w1 AND "Blend_T-20".State."BFT-1 EN" THEN
       #"P-20.01".IN_SP_Speed := "Blend_T-20".Out_P_Transfer1_Sp;
   END_IF;
   IF #_w1 AND "Blend_T-21".State."BFT-1 EN" THEN
       #"P-20.01".IN_SP_Speed := "Blend_T-21".Out_P_Transfer1_Sp;
   END_IF;
   IF #_w1 AND "Blend_T-30".State."BFT-1 EN" THEN
       #"P-20.01".IN_SP_Speed := "Blend_T-30".Out_P_Transfer1_Sp;
   END_IF;
   IF #_w1 AND "General_Blend".Blend_Cluster1.CIP_Line1."CIP Request" THEN
       #"P-20.01".IN_SP_Speed := "General_Blend".Blend_Cluster1.CIP_Line1.P_SP;
   END_IF;
   IF "AlwaysTRUE" AND NOT #"P-20.01".QMAN_AUT THEN #"P-20.01".IN_SP_Speed := #"P-20.01".IN_SP_Speed; END_IF;
END_REGION

REGION Network 23: P-20.01
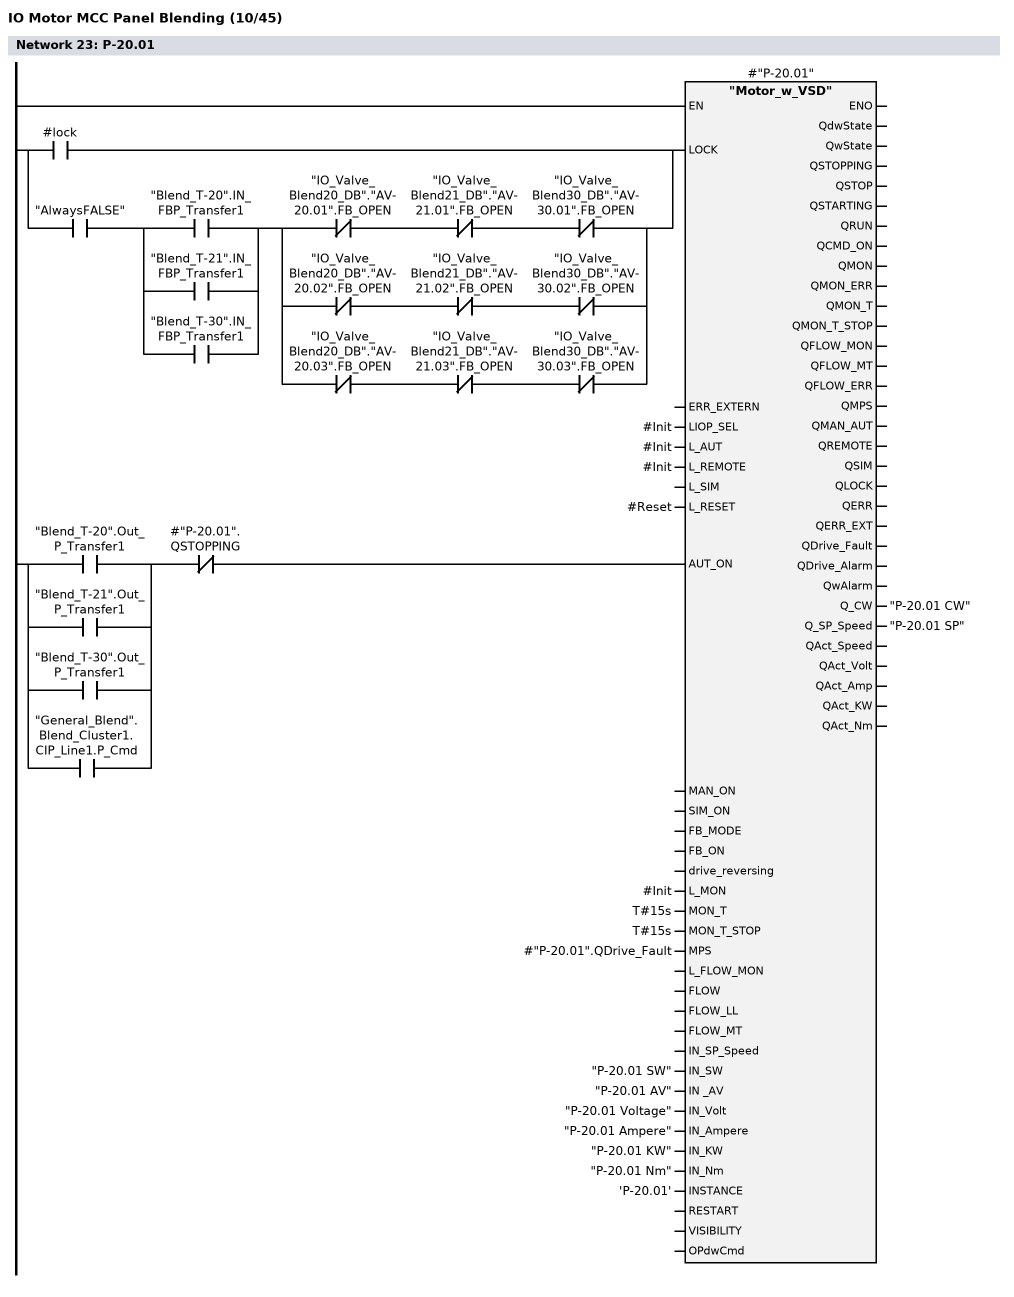
   RUNG wire#powerrail
      #"P-20.01"(LOCK := wire#w3, AUT_ON := wire#w5, ERR_EXTERN :=, LIOP_SEL := #Init, L_AUT := #Init, L_REMOTE := #Init, L_SIM :=, L_RESET := #Reset, MAN_ON :=, SIM_ON :=, FB_MODE :=, FB_ON :=, drive_reversing :=, L_MON := #Init, MON_T := T#15s, MON_T_STOP := T#15s, MPS := #"P-20.01".QDrive_Fault, L_FLOW_MON :=, FLOW :=, FLOW_LL :=, FLOW_MT :=, IN_SP_Speed :=, IN_SW := "P-20.01 SW", "IN _AV" := "P-20.01 AV", IN_Volt := "P-20.01 Voltage", IN_Ampere := "P-20.01 Ampere", IN_KW := "P-20.01 KW", IN_Nm := "P-20.01 Nm", INSTANCE := 'P-20.01', RESTART :=, VISIBILITY :=, OPdwCmd :=, QdwState =>, QwState =>, QSTOPPING =>, QSTOP =>, QSTARTING =>, QRUN =>, QCMD_ON =>, QMON =>, QMON_ERR =>, QMON_T =>, QMON_T_STOP =>, QFLOW_MON =>, QFLOW_MT =>, QFLOW_ERR =>, QMPS =>, QMAN_AUT =>, QREMOTE =>, QSIM =>, QLOCK =>, QERR =>, QERR_EXT =>, QDrive_Fault =>, QDrive_Alarm =>, QwAlarm =>, Q_CW => "P-20.01 CW", Q_SP_Speed => "P-20.01 SP", QAct_Speed =>, QAct_Volt =>, QAct_Amp =>, QAct_KW =>, QAct_Nm =>)
   END_RUNG
   RUNG wire#powerrail
      Contact( #lock )
   END_RUNG wire#w3
   RUNG wire#powerrail
      Contact( "AlwaysFALSE" )
      wire#w1
      Contact( "Blend_T-20".IN_FBP_Transfer1 )
      wire#w2
      I_Contact( "IO_Valve_Blend20_DB"."AV-20.01".FB_OPEN )
      I_Contact( "IO_Valve_Blend21_DB"."AV-21.01".FB_OPEN )
      I_Contact( "IO_Valve_Blend30_DB"."AV-30.01".FB_OPEN )
   END_RUNG wire#w3
   RUNG wire#w1
      Contact( "Blend_T-21".IN_FBP_Transfer1 )
   END_RUNG wire#w2
   RUNG wire#w1
      Contact( "Blend_T-30".IN_FBP_Transfer1 )
   END_RUNG wire#w2
   RUNG wire#w2
      I_Contact( "IO_Valve_Blend20_DB"."AV-20.02".FB_OPEN )
      I_Contact( "IO_Valve_Blend21_DB"."AV-21.02".FB_OPEN )
      I_Contact( "IO_Valve_Blend30_DB"."AV-30.02".FB_OPEN )
   END_RUNG wire#w3
   RUNG wire#w2
      I_Contact( "IO_Valve_Blend20_DB"."AV-20.03".FB_OPEN )
      I_Contact( "IO_Valve_Blend21_DB"."AV-21.03".FB_OPEN )
      I_Contact( "IO_Valve_Blend30_DB"."AV-30.03".FB_OPEN )
   END_RUNG wire#w3
   RUNG wire#powerrail
      Contact( "Blend_T-20".Out_P_Transfer1 )
      wire#w4
      I_Contact( #"P-20.01".QSTOPPING )
   END_RUNG wire#w5
   RUNG wire#powerrail
      Contact( "Blend_T-21".Out_P_Transfer1 )
   END_RUNG wire#w4
   RUNG wire#powerrail
      Contact( "Blend_T-30".Out_P_Transfer1 )
   END_RUNG wire#w4
   RUNG wire#powerrail
      Contact( "General_Blend".Blend_Cluster1.CIP_Line1.P_Cmd )
   END_RUNG wire#w4
   // the same network as SCL:
   #"P-20.01"(LOCK := #lock OR ("AlwaysFALSE" AND ("Blend_T-20".IN_FBP_Transfer1 OR "Blend_T-21".IN_FBP_Transfer1 OR "Blend_T-30".IN_FBP_Transfer1) AND ((NOT "IO_Valve_Blend20_DB"."AV-20.01".FB_OPEN AND NOT "IO_Valve_Blend21_DB"."AV-21.01".FB_OPEN AND NOT "IO_Valve_Blend30_DB"."AV-30.01".FB_OPEN) OR (NOT "IO_Valve_Blend20_DB"."AV-20.02".FB_OPEN AND NOT "IO_Valve_Blend21_DB"."AV-21.02".FB_OPEN AND NOT "IO_Valve_Blend30_DB"."AV-30.02".FB_OPEN) OR (NOT "IO_Valve_Blend20_DB"."AV-20.03".FB_OPEN AND NOT "IO_Valve_Blend21_DB"."AV-21.03".FB_OPEN AND NOT "IO_Valve_Blend30_DB"."AV-30.03".FB_OPEN))),   // "Motor_w_VSD"
              LIOP_SEL := #Init,
              L_AUT := #Init,
              L_REMOTE := #Init,
              L_RESET := #Reset,
              AUT_ON := ("Blend_T-20".Out_P_Transfer1 OR "Blend_T-21".Out_P_Transfer1 OR "Blend_T-30".Out_P_Transfer1 OR "General_Blend".Blend_Cluster1.CIP_Line1.P_Cmd) AND NOT #"P-20.01".QSTOPPING,
              L_MON := #Init,
              MON_T := T#15s,
              MON_T_STOP := T#15s,
              MPS := #"P-20.01".QDrive_Fault,
              IN_SW := "P-20.01 SW",
              "IN _AV" := "P-20.01 AV",
              IN_Volt := "P-20.01 Voltage",
              IN_Ampere := "P-20.01 Ampere",
              IN_KW := "P-20.01 KW",
              IN_Nm := "P-20.01 Nm",
              INSTANCE := 'P-20.01',
              Q_CW => "P-20.01 CW",
              Q_SP_Speed => "P-20.01 SP");
END_REGION

REGION Network 24: P-21.01 Speed
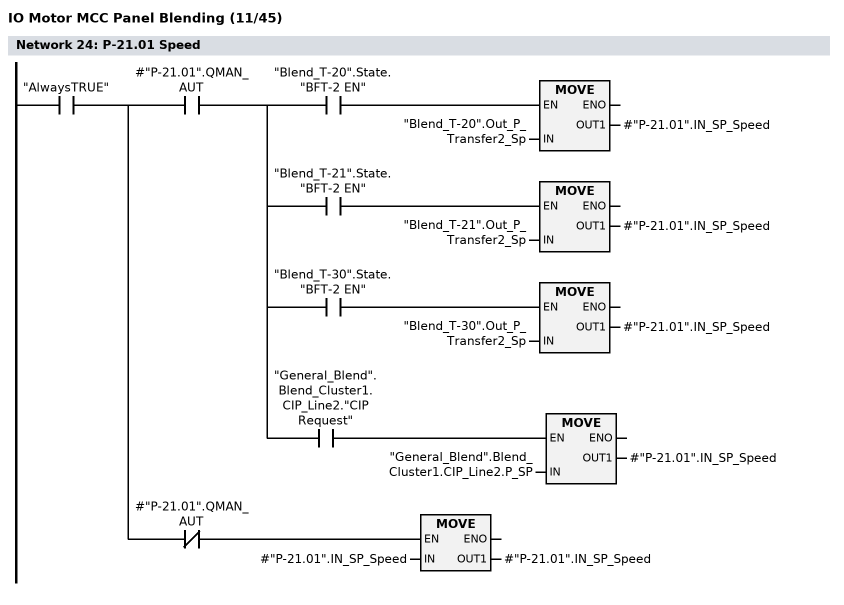
   RUNG wire#powerrail
      Contact( "AlwaysTRUE" )
      wire#w1
      Contact( #"P-21.01".QMAN_AUT )
      wire#w2
      Contact( "Blend_T-20".State."BFT-2 EN" )
      Move(in := "Blend_T-20".Out_P_Transfer2_Sp, out1 => #"P-21.01".IN_SP_Speed)
   END_RUNG
   RUNG wire#w2
      Contact( "Blend_T-21".State."BFT-2 EN" )
      Move(in := "Blend_T-21".Out_P_Transfer2_Sp, out1 => #"P-21.01".IN_SP_Speed)
   END_RUNG
   RUNG wire#w2
      Contact( "Blend_T-30".State."BFT-2 EN" )
      Move(in := "Blend_T-30".Out_P_Transfer2_Sp, out1 => #"P-21.01".IN_SP_Speed)
   END_RUNG
   RUNG wire#w2
      Contact( "General_Blend".Blend_Cluster1.CIP_Line2."CIP Request" )
      Move(in := "General_Blend".Blend_Cluster1.CIP_Line2.P_SP, out1 => #"P-21.01".IN_SP_Speed)
   END_RUNG
   RUNG wire#w1
      I_Contact( #"P-21.01".QMAN_AUT )
      Move(in := #"P-21.01".IN_SP_Speed, out1 => #"P-21.01".IN_SP_Speed)
   END_RUNG
   // the same network as SCL:
   #_w1 := "AlwaysTRUE" AND #"P-21.01".QMAN_AUT;
   IF #_w1 AND "Blend_T-20".State."BFT-2 EN" THEN
       #"P-21.01".IN_SP_Speed := "Blend_T-20".Out_P_Transfer2_Sp;
   END_IF;
   IF #_w1 AND "Blend_T-21".State."BFT-2 EN" THEN
       #"P-21.01".IN_SP_Speed := "Blend_T-21".Out_P_Transfer2_Sp;
   END_IF;
   IF #_w1 AND "Blend_T-30".State."BFT-2 EN" THEN
       #"P-21.01".IN_SP_Speed := "Blend_T-30".Out_P_Transfer2_Sp;
   END_IF;
   IF #_w1 AND "General_Blend".Blend_Cluster1.CIP_Line2."CIP Request" THEN
       #"P-21.01".IN_SP_Speed := "General_Blend".Blend_Cluster1.CIP_Line2.P_SP;
   END_IF;
   IF "AlwaysTRUE" AND NOT #"P-21.01".QMAN_AUT THEN #"P-21.01".IN_SP_Speed := #"P-21.01".IN_SP_Speed; END_IF;
END_REGION

REGION Network 25: P-21.01
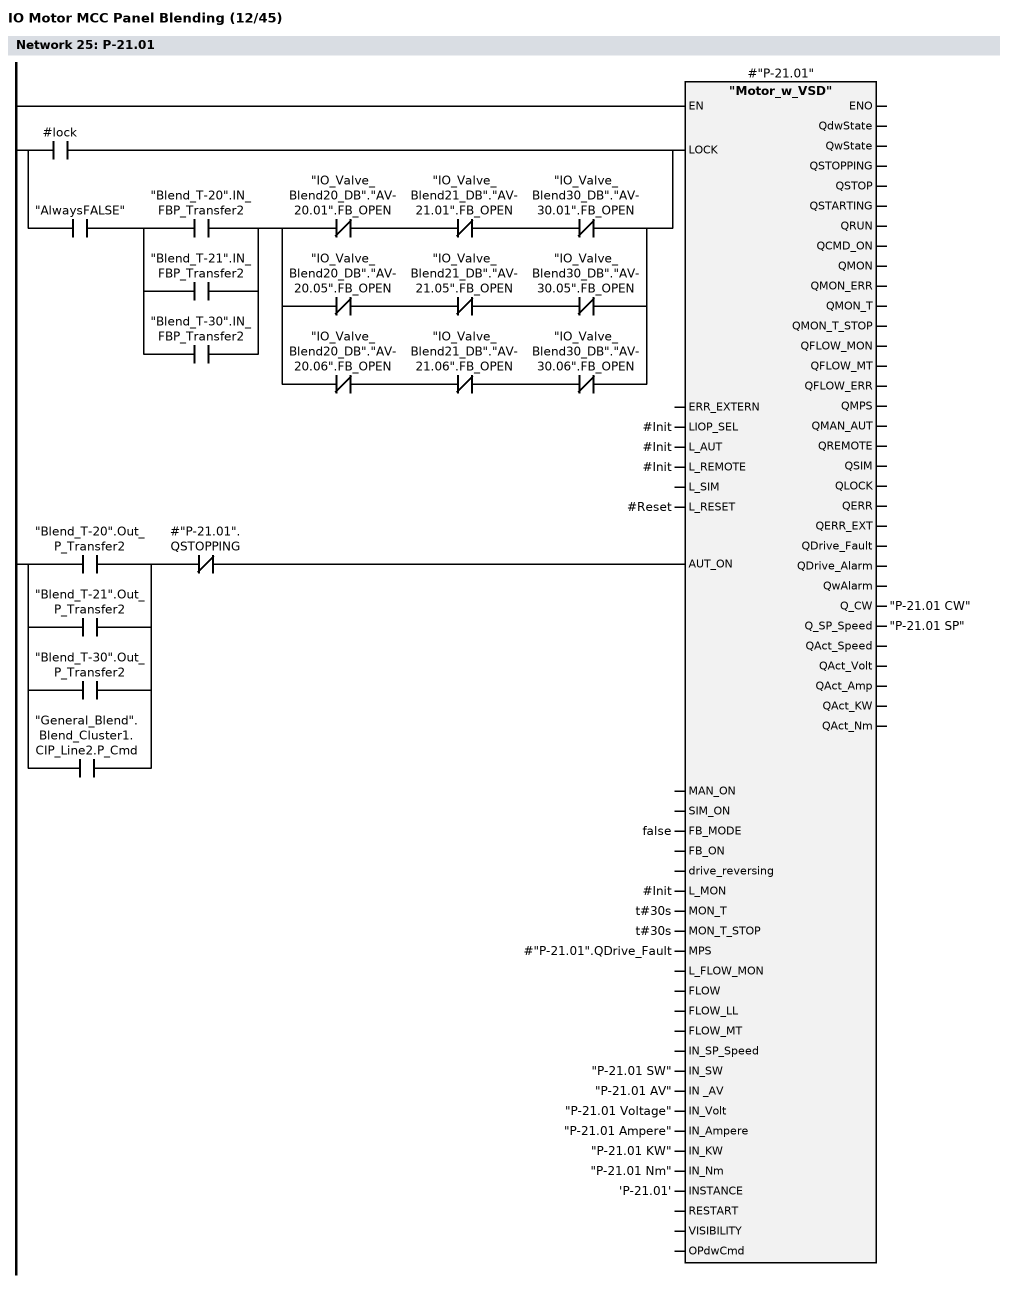
   RUNG wire#powerrail
      #"P-21.01"(LOCK := wire#w3, AUT_ON := wire#w5, ERR_EXTERN :=, LIOP_SEL := #Init, L_AUT := #Init, L_REMOTE := #Init, L_SIM :=, L_RESET := #Reset, MAN_ON :=, SIM_ON :=, FB_MODE := false, FB_ON :=, drive_reversing :=, L_MON := #Init, MON_T := t#30s, MON_T_STOP := t#30s, MPS := #"P-21.01".QDrive_Fault, L_FLOW_MON :=, FLOW :=, FLOW_LL :=, FLOW_MT :=, IN_SP_Speed :=, IN_SW := "P-21.01 SW", "IN _AV" := "P-21.01 AV", IN_Volt := "P-21.01 Voltage", IN_Ampere := "P-21.01 Ampere", IN_KW := "P-21.01 KW", IN_Nm := "P-21.01 Nm", INSTANCE := 'P-21.01', RESTART :=, VISIBILITY :=, OPdwCmd :=, QdwState =>, QwState =>, QSTOPPING =>, QSTOP =>, QSTARTING =>, QRUN =>, QCMD_ON =>, QMON =>, QMON_ERR =>, QMON_T =>, QMON_T_STOP =>, QFLOW_MON =>, QFLOW_MT =>, QFLOW_ERR =>, QMPS =>, QMAN_AUT =>, QREMOTE =>, QSIM =>, QLOCK =>, QERR =>, QERR_EXT =>, QDrive_Fault =>, QDrive_Alarm =>, QwAlarm =>, Q_CW => "P-21.01 CW", Q_SP_Speed => "P-21.01 SP", QAct_Speed =>, QAct_Volt =>, QAct_Amp =>, QAct_KW =>, QAct_Nm =>)
   END_RUNG
   RUNG wire#powerrail
      Contact( #lock )
   END_RUNG wire#w3
   RUNG wire#powerrail
      Contact( "AlwaysFALSE" )
      wire#w1
      Contact( "Blend_T-20".IN_FBP_Transfer2 )
      wire#w2
      I_Contact( "IO_Valve_Blend20_DB"."AV-20.01".FB_OPEN )
      I_Contact( "IO_Valve_Blend21_DB"."AV-21.01".FB_OPEN )
      I_Contact( "IO_Valve_Blend30_DB"."AV-30.01".FB_OPEN )
   END_RUNG wire#w3
   RUNG wire#w1
      Contact( "Blend_T-21".IN_FBP_Transfer2 )
   END_RUNG wire#w2
   RUNG wire#w1
      Contact( "Blend_T-30".IN_FBP_Transfer2 )
   END_RUNG wire#w2
   RUNG wire#w2
      I_Contact( "IO_Valve_Blend20_DB"."AV-20.05".FB_OPEN )
      I_Contact( "IO_Valve_Blend21_DB"."AV-21.05".FB_OPEN )
      I_Contact( "IO_Valve_Blend30_DB"."AV-30.05".FB_OPEN )
   END_RUNG wire#w3
   RUNG wire#w2
      I_Contact( "IO_Valve_Blend20_DB"."AV-20.06".FB_OPEN )
      I_Contact( "IO_Valve_Blend21_DB"."AV-21.06".FB_OPEN )
      I_Contact( "IO_Valve_Blend30_DB"."AV-30.06".FB_OPEN )
   END_RUNG wire#w3
   RUNG wire#powerrail
      Contact( "Blend_T-20".Out_P_Transfer2 )
      wire#w4
      I_Contact( #"P-21.01".QSTOPPING )
   END_RUNG wire#w5
   RUNG wire#powerrail
      Contact( "Blend_T-21".Out_P_Transfer2 )
   END_RUNG wire#w4
   RUNG wire#powerrail
      Contact( "Blend_T-30".Out_P_Transfer2 )
   END_RUNG wire#w4
   RUNG wire#powerrail
      Contact( "General_Blend".Blend_Cluster1.CIP_Line2.P_Cmd )
   END_RUNG wire#w4
   // the same network as SCL:
   #"P-21.01"(LOCK := #lock OR ("AlwaysFALSE" AND ("Blend_T-20".IN_FBP_Transfer2 OR "Blend_T-21".IN_FBP_Transfer2 OR "Blend_T-30".IN_FBP_Transfer2) AND ((NOT "IO_Valve_Blend20_DB"."AV-20.01".FB_OPEN AND NOT "IO_Valve_Blend21_DB"."AV-21.01".FB_OPEN AND NOT "IO_Valve_Blend30_DB"."AV-30.01".FB_OPEN) OR (NOT "IO_Valve_Blend20_DB"."AV-20.05".FB_OPEN AND NOT "IO_Valve_Blend21_DB"."AV-21.05".FB_OPEN AND NOT "IO_Valve_Blend30_DB"."AV-30.05".FB_OPEN) OR (NOT "IO_Valve_Blend20_DB"."AV-20.06".FB_OPEN AND NOT "IO_Valve_Blend21_DB"."AV-21.06".FB_OPEN AND NOT "IO_Valve_Blend30_DB"."AV-30.06".FB_OPEN))),   // "Motor_w_VSD"
              LIOP_SEL := #Init,
              L_AUT := #Init,
              L_REMOTE := #Init,
              L_RESET := #Reset,
              AUT_ON := ("Blend_T-20".Out_P_Transfer2 OR "Blend_T-21".Out_P_Transfer2 OR "Blend_T-30".Out_P_Transfer2 OR "General_Blend".Blend_Cluster1.CIP_Line2.P_Cmd) AND NOT #"P-21.01".QSTOPPING,
              FB_MODE := false,
              L_MON := #Init,
              MON_T := t#30s,
              MON_T_STOP := t#30s,
              MPS := #"P-21.01".QDrive_Fault,
              IN_SW := "P-21.01 SW",
              "IN _AV" := "P-21.01 AV",
              IN_Volt := "P-21.01 Voltage",
              IN_Ampere := "P-21.01 Ampere",
              IN_KW := "P-21.01 KW",
              IN_Nm := "P-21.01 Nm",
              INSTANCE := 'P-21.01',
              Q_CW => "P-21.01 CW",
              Q_SP_Speed => "P-21.01 SP");
END_REGION

REGION Network 26: P-30.01 Speed
